C03584=1030.915,110.393,-100.515,168.841,44.081,158.264
C03585=1030.909,110.144,-100.496,168.839,44.083,158.265
C03586=1030.902,109.895,-100.475,168.837,44.085,158.265
C03587=1030.896,109.646,-100.456,168.834,44.087,158.265
C03588=1030.890,109.397,-100.436,168.831,44.089,158.265
C03589=1030.884,109.148,-100.417,168.829,44.091,158.265
C03590=1030.878,108.899,-100.397,168.826,44.093,158.265
C03591=1030.870,108.613,-100.375,168.824,44.095,158.265
C03592=1030.864,108.328,-100.352,168.821,44.097,158.266
C03593=1030.857,108.042,-100.330,168.818,44.099,158.266
C03594=1030.850,107.758,-100.307,168.815,44.101,158.266
C03595=1030.844,107.508,-100.288,168.812,44.103,158.266
C03596=1030.837,107.259,-100.268,168.811,44.105,158.266
C03597=1030.831,107.010,-100.249,168.808,44.107,158.266
C03598=1030.825,106.761,-100.229,168.806,44.109,158.267
C03599=1030.819,106.511,-100.210,168.803,44.110,158.267
C03600=1030.813,106.263,-100.191,168.800,44.112,158.267
C03601=1030.807,106.013,-100.171,168.798,44.114,158.267
C03602=1030.800,105.764,-100.151,168.795,44.115,158.267
C03603=1030.795,105.515,-100.132,168.793,44.117,158.267
C03604=1030.788,105.265,-100.113,168.791,44.119,158.267
C03605=1030.782,105.017,-100.093,168.788,44.121,158.267
C03606=1030.776,104.767,-100.074,168.786,44.123,158.268
C03607=1030.770,104.518,-100.054,168.783,44.125,158.268
C03608=1030.764,104.269,-100.035,168.781,44.127,158.268
C03609=1030.758,104.020,-100.015,168.779,44.128,158.268
C03610=1030.752,103.770,-99.996,168.776,44.130,158.268
C03611=1030.745,103.521,-99.977,168.774,44.132,158.268
C03612=1030.739,103.272,-99.957,168.771,44.134,158.268
C03613=1030.734,103.023,-99.938,168.768,44.135,158.268
C03614=1030.728,102.774,-99.918,168.767,44.137,158.269
C03615=1030.721,102.525,-99.899,168.764,44.139,158.269
C03616=1030.716,102.276,-99.880,168.762,44.141,158.269
C03617=1030.710,102.027,-99.860,168.759,44.143,158.269
C03618=1030.704,101.777,-99.841,168.756,44.145,158.269
C03619=1030.697,101.528,-99.822,168.755,44.146,158.269
C03620=1030.691,101.279,-99.802,168.752,44.148,158.269
C03621=1030.686,101.030,-99.783,168.749,44.150,158.269
C03622=1030.679,100.781,-99.764,168.747,44.151,158.270
C03623=1030.673,100.531,-99.744,168.744,44.153,158.270
C03624=1030.667,100.282,-99.725,168.743,44.155,158.270
C03625=1030.661,100.032,-99.706,168.740,44.157,158.270
C03626=1030.655,99.784,-99.686,168.737,44.159,158.270
C03627=1030.649,99.534,-99.667,168.735,44.161,158.270
C03628=1030.643,99.285,-99.648,168.732,44.163,158.270
C03629=1030.637,99.036,-99.629,168.730,44.165,158.271
C03630=1030.630,98.787,-99.610,168.728,44.166,158.271
C03631=1030.625,98.537,-99.591,168.726,44.168,158.271
C03632=1030.618,98.289,-99.572,168.723,44.170,158.271
C03633=1030.612,98.040,-99.553,168.720,44.172,158.271
C03634=1030.606,97.790,-99.534,168.718,44.174,158.271
C03635=1030.599,97.541,-99.515,168.715,44.176,158.271
C03636=1030.594,97.292,-99.496,168.714,44.178,158.272
C03637=1030.587,97.043,-99.477,168.711,44.180,158.272
C03638=1030.581,96.794,-99.457,168.708,44.181,158.272
C03639=1030.575,96.545,-99.439,168.706,44.183,158.272
C03640=1030.569,96.295,-99.420,168.703,44.185,158.272
C03641=1030.563,96.046,-99.401,168.701,44.187,158.272
C03642=1030.556,95.797,-99.382,168.699,44.189,158.273
C03643=1030.551,95.548,-99.363,168.696,44.191,158.273
C03644=1030.544,95.298,-99.344,168.694,44.193,158.273
C03645=1030.539,95.049,-99.325,168.691,44.195,158.273
C03646=1030.532,94.800,-99.306,168.689,44.197,158.273
C03647=1030.526,94.550,-99.287,168.687,44.198,158.273
C03648=1030.520,94.301,-99.269,168.684,44.200,158.273
C03649=1030.514,94.053,-99.249,168.682,44.202,158.274
C03650=1030.508,93.803,-99.230,168.679,44.204,158.274
C03651=1030.501,93.554,-99.211,168.677,44.206,158.274
C03652=1030.496,93.305,-99.192,168.675,44.208,158.274
C03653=1030.489,93.056,-99.173,168.673,44.210,158.274
C03654=1030.483,92.806,-99.154,168.670,44.211,158.274
C03655=1030.476,92.521,-99.134,168.667,44.213,158.274
C03656=1030.469,92.236,-99.112,168.665,44.215,158.275
C03657=1030.462,91.950,-99.089,168.661,44.217,158.275
C03658=1030.455,91.665,-99.068,168.659,44.219,158.275
C03659=1030.449,91.416,-99.049,168.656,44.221,158.275
C03660=1030.443,91.166,-99.030,168.654,44.223,158.275
C03661=1030.437,90.918,-99.012,168.652,44.225,158.275
C03662=1030.431,90.669,-98.993,168.649,44.227,158.275
C03663=1030.425,90.419,-98.974,168.647,44.229,158.275
C03664=1030.419,90.170,-98.955,168.644,44.231,158.276
C03665=1030.413,89.921,-98.936,168.642,44.232,158.276
C03666=1030.407,89.672,-98.917,168.640,44.234,158.276
C03667=1030.400,89.422,-98.899,168.637,44.236,158.276
C03668=1030.394,89.173,-98.881,168.635,44.238,158.276
C03669=1030.388,88.923,-98.862,168.632,44.240,158.276
C03670=1030.382,88.674,-98.843,168.631,44.242,158.277
C03671=1030.376,88.425,-98.824,168.628,44.244,158.277
C03672=1030.369,88.176,-98.806,168.625,44.245,158.277
C03673=1030.363,87.926,-98.788,168.623,44.247,158.277
C03674=1030.357,87.677,-98.769,168.620,44.249,158.277
C03675=1030.351,87.429,-98.751,168.618,44.252,158.277
C03676=1030.345,87.179,-98.731,168.616,44.254,158.278
C03677=1030.339,86.929,-98.714,168.614,44.256,158.278
C03678=1030.333,86.680,-98.695,168.611,44.257,158.278
C03679=1030.326,86.431,-98.676,168.608,44.259,158.278
C03680=1030.320,86.182,-98.658,168.606,44.261,158.278
C03681=1030.314,85.932,-98.640,168.604,44.263,158.278
C03682=1030.307,85.683,-98.621,168.602,44.265,158.278
C03683=1030.301,85.434,-98.602,168.599,44.267,158.279
C03684=1030.296,85.185,-98.583,168.597,44.269,158.279
C03685=1030.290,84.936,-98.566,168.594,44.271,158.279
C03686=1030.283,84.686,-98.547,168.591,44.273,158.279
C03687=1030.277,84.437,-98.528,168.590,44.274,158.279
C03688=1030.271,84.188,-98.510,168.587,44.276,158.279
C03689=1030.264,83.938,-98.492,168.585,44.278,158.279
C03690=1030.258,83.689,-98.473,168.582,44.280,158.280
C03691=1030.252,83.441,-98.455,168.579,44.282,158.280
C03692=1030.246,83.191,-98.437,168.578,44.284,158.280
C03693=1030.240,82.942,-98.418,168.575,44.286,158.280
C03694=1030.234,82.693,-98.399,168.573,44.288,158.280
C03695=1030.228,82.443,-98.381,168.570,44.290,158.280
C03696=1030.222,82.194,-98.363,168.567,44.291,158.280
C03697=1030.216,81.945,-98.345,168.566,44.293,158.281
C03698=1030.209,81.696,-98.326,168.563,44.295,158.281
C03699=1030.203,81.446,-98.307,168.561,44.297,158.281
C03700=1030.197,81.197,-98.290,168.558,44.299,158.281
C03701=1030.191,80.948,-98.271,168.557,44.301,158.281
C03702=1030.185,80.698,-98.253,168.554,44.303,158.281
C03703=1030.179,80.449,-98.234,168.551,44.304,158.281
C03704=1030.173,80.200,-98.215,168.549,44.306,158.282
C03705=1030.166,79.950,-98.197,168.546,44.308,158.282
C03706=1030.161,79.702,-98.179,168.545,44.310,158.282
C03707=1030.155,79.452,-98.161,168.542,44.312,158.282
C03708=1030.148,79.203,-98.143,168.539,44.314,158.282
C03709=1030.142,78.953,-98.125,168.537,44.316,158.282
C03710=1030.136,78.705,-98.106,168.535,44.318,158.282
C03711=1030.130,78.456,-98.088,168.533,44.319,158.283
C03712=1030.124,78.206,-98.070,168.530,44.321,158.283
C03713=1030.118,77.957,-98.051,168.528,44.323,158.283
C03714=1030.112,77.708,-98.033,168.525,44.325,158.283
C03715=1030.106,77.458,-98.016,168.523,44.327,158.283
C03716=1030.099,77.209,-97.997,168.521,44.329,158.283
C03717=1030.093,76.959,-97.979,168.518,44.331,158.283
C03718=1030.087,76.711,-97.961,168.516,44.333,158.284
C03719=1030.080,76.425,-97.940,168.513,44.335,158.284
C03720=1030.073,76.140,-97.919,168.511,44.337,158.284
C03721=1030.066,75.855,-97.898,168.508,44.339,158.284
C03722=1030.059,75.569,-97.878,168.505,44.342,158.284
C03723=1030.053,75.320,-97.860,168.503,44.344,158.284
C03724=1030.046,75.070,-97.842,168.501,44.346,158.285
C03725=1030.040,74.821,-97.825,168.498,44.348,158.285
C03726=1030.034,74.572,-97.806,168.495,44.349,158.285
C03727=1030.028,74.322,-97.788,168.493,44.351,158.285
C03728=1030.022,74.073,-97.771,168.490,44.353,158.285
C03729=1030.016,73.824,-97.752,168.489,44.355,158.285
C03730=1030.009,73.575,-97.735,168.486,44.357,158.285
C03731=1030.003,73.325,-97.717,168.483,44.359,158.286
C03732=1029.997,73.076,-97.698,168.481,44.361,158.286
C03733=1029.991,72.827,-97.680,168.478,44.363,158.286
C03734=1029.985,72.577,-97.662,168.477,44.365,158.286
C03735=1029.978,72.329,-97.645,168.474,44.366,158.286
C03736=1029.972,72.079,-97.627,168.471,44.368,158.286
C03737=1029.966,71.829,-97.609,168.469,44.370,158.286
C03738=1029.960,71.580,-97.591,168.466,44.372,158.287
C03739=1029.954,71.331,-97.573,168.465,44.374,158.287
C03740=1029.947,71.082,-97.555,168.462,44.376,158.287
C03741=1029.942,70.833,-97.538,168.460,44.378,158.287
C03742=1029.936,70.583,-97.520,168.457,44.380,158.287
C03743=1029.929,70.334,-97.501,168.456,44.382,158.287
C03744=1029.924,70.085,-97.484,168.453,44.384,158.288
C03745=1029.917,69.835,-97.466,168.450,44.386,158.288
C03746=1029.911,69.586,-97.448,168.448,44.388,158.288
C03747=1029.905,69.337,-97.431,168.445,44.390,158.288
C03748=1029.899,69.087,-97.412,168.444,44.392,158.288
C03749=1029.892,68.838,-97.395,168.441,44.394,158.288
C03750=1029.886,68.589,-97.377,168.439,44.395,158.288
C03751=1029.880,68.339,-97.359,168.436,44.397,158.289
C03752=1029.874,68.091,-97.342,168.433,44.399,158.289
C03753=1029.868,67.841,-97.324,168.432,44.401,158.289
C03754=1029.862,67.591,-97.306,168.429,44.403,158.289
C03755=1029.855,67.343,-97.289,168.427,44.405,158.289
C03756=1029.849,67.093,-97.271,168.424,44.407,158.289
C03757=1029.842,66.844,-97.254,168.421,44.409,158.289
C03758=1029.837,66.595,-97.236,168.419,44.411,158.290
C03759=1029.831,66.345,-97.218,168.418,44.413,158.290
C03760=1029.824,66.096,-97.201,168.415,44.415,158.290
C03761=1029.818,65.847,-97.183,168.412,44.417,158.290
C03762=1029.811,65.597,-97.166,168.410,44.419,158.290
C03763=1029.806,65.348,-97.148,168.407,44.421,158.290
C03764=1029.800,65.098,-97.130,168.406,44.423,158.290
C03765=1029.793,64.850,-97.113,168.403,44.424,158.291
C03766=1029.787,64.600,-97.095,168.400,44.426,158.291
C03767=1029.781,64.351,-97.078,168.398,44.428,158.291
C03768=1029.775,64.101,-97.060,168.395,44.430,158.291
C03769=1029.768,63.852,-97.043,168.394,44.432,158.291
C03770=1029.763,63.603,-97.026,168.391,44.434,158.291
C03771=1029.756,63.353,-97.008,168.389,44.437,158.292
C03772=1029.750,63.104,-96.991,168.386,44.439,158.292
C03773=1029.743,62.855,-96.973,168.384,44.440,158.292
C03774=1029.736,62.606,-96.956,168.381,44.442,158.292
C03775=1029.731,62.356,-96.939,168.379,44.445,158.292
C03776=1029.724,62.106,-96.922,168.377,44.447,158.292
C03777=1029.718,61.858,-96.905,168.374,44.449,158.293
C03778=1029.712,61.608,-96.887,168.372,44.451,158.293
C03779=1029.706,61.359,-96.870,168.369,44.453,158.293
C03780=1029.699,61.110,-96.853,168.367,44.455,158.293
C03781=1029.692,60.860,-96.836,168.364,44.457,158.293
C03782=1029.687,60.611,-96.818,168.362,44.459,158.293
C03783=1029.679,60.325,-96.799,168.359,44.462,158.294
C03784=1029.672,60.040,-96.778,168.357,44.464,158.294
C03785=1029.665,59.755,-96.759,168.354,44.466,158.294
C03786=1029.658,59.469,-96.739,168.351,44.468,158.294
C03787=1029.651,59.220,-96.722,168.348,44.470,158.294
C03788=1029.645,58.970,-96.706,168.347,44.472,158.294
C03789=1029.639,58.720,-96.688,168.344,44.475,158.295
C03790=1029.633,58.472,-96.671,168.342,44.477,158.295
C03791=1029.626,58.222,-96.654,168.339,44.478,158.295
C03792=1029.620,57.973,-96.637,168.337,44.480,158.295
C03793=1029.614,57.723,-96.619,168.334,44.482,158.295
C03794=1029.607,57.475,-96.602,168.332,44.484,158.295
C03795=1029.601,57.225,-96.585,168.330,44.487,158.296
C03796=1029.595,56.975,-96.568,168.328,44.489,158.296
C03797=1029.588,56.726,-96.551,168.325,44.491,158.296
C03798=1029.582,56.477,-96.534,168.322,44.492,158.296
C03799=1029.576,56.227,-96.517,168.320,44.494,158.296
C03800=1029.570,55.978,-96.500,168.318,44.496,158.296
C03801=1029.563,55.729,-96.482,168.316,44.498,158.296
C03802=1029.557,55.479,-96.466,168.313,44.501,158.297
C03803=1029.550,55.230,-96.449,168.311,44.503,158.297
C03804=1029.545,54.981,-96.431,168.308,44.505,158.297
C03805=1029.538,54.731,-96.415,168.305,44.507,158.297
C03806=1029.532,54.482,-96.398,168.303,44.508,158.297
C03807=1029.526,54.233,-96.381,168.301,44.510,158.297
C03808=1029.520,53.983,-96.363,168.299,44.512,158.297
C03809=1029.514,53.734,-96.346,168.296,44.514,158.298
C03810=1029.507,53.485,-96.329,168.294,44.517,158.298
C03811=1029.502,53.235,-96.312,168.291,44.519,158.298
C03812=1029.495,52.986,-96.295,168.290,44.520,158.298
C03813=1029.489,52.736,-96.279,168.287,44.522,158.298
C03814=1029.483,52.488,-96.262,168.284,44.524,158.298
C03815=1029.477,52.238,-96.244,168.282,44.526,158.299
C03816=1029.471,51.989,-96.228,168.279,44.528,158.299
C03817=1029.464,51.739,-96.210,168.277,44.530,158.299
C03818=1029.458,51.490,-96.194,168.275,44.532,158.299
C03819=1029.452,51.241,-96.177,168.273,44.534,158.299
C03820=1029.446,50.991,-96.160,168.270,44.536,158.299
C03821=1029.439,50.742,-96.143,168.268,44.538,158.300
C03822=1029.433,50.493,-96.127,168.265,44.540,158.300
C03823=1029.427,50.243,-96.109,168.262,44.542,158.300
C03824=1029.421,49.994,-96.092,168.261,44.544,158.300
C03825=1029.415,49.744,-96.075,168.258,44.546,158.300
C03826=1029.408,49.495,-96.058,168.256,44.548,158.300
C03827=1029.402,49.246,-96.042,168.253,44.550,158.300
C03828=1029.396,48.996,-96.024,168.251,44.552,158.300
C03829=1029.390,48.747,-96.008,168.249,44.554,158.301
C03830=1029.384,48.498,-95.991,168.246,44.555,158.301
C03831=1029.377,48.248,-95.974,168.244,44.557,158.301
C03832=1029.372,47.999,-95.957,168.241,44.559,158.301
C03833=1029.366,47.750,-95.940,168.239,44.561,158.301
C03834=1029.360,47.500,-95.924,168.237,44.563,158.301
C03835=1029.353,47.251,-95.907,168.235,44.565,158.301
C03836=1029.347,47.002,-95.890,168.232,44.567,158.302
C03837=1029.342,46.753,-95.873,168.229,44.569,158.302
C03838=1029.335,46.503,-95.856,168.227,44.571,158.302
C03839=1029.329,46.254,-95.839,168.225,44.573,158.302
C03840=1029.323,46.005,-95.823,168.223,44.575,158.302
C03841=1029.317,45.754,-95.806,168.220,44.576,158.302
C03842=1029.311,45.505,-95.789,168.217,44.578,158.302
C03843=1029.305,45.256,-95.772,168.215,44.580,158.302
C03844=1029.299,45.007,-95.755,168.213,44.582,158.303
C03845=1029.292,44.757,-95.739,168.211,44.584,158.303
C03846=1029.287,44.508,-95.722,168.208,44.586,158.303
C03847=1029.279,44.222,-95.703,168.206,44.588,158.303
C03848=1029.273,43.936,-95.684,168.203,44.591,158.303
C03849=1029.265,43.651,-95.664,168.200,44.593,158.303
C03850=1029.259,43.365,-95.646,168.197,44.595,158.303
C03851=1029.253,43.115,-95.628,168.194,44.597,158.304
C03852=1029.247,42.866,-95.612,168.193,44.598,158.304
C03853=1029.241,42.617,-95.596,168.190,44.600,158.304
C03854=1029.235,42.367,-95.579,168.188,44.602,158.304
C03855=1029.228,42.118,-95.562,168.185,44.604,158.304
C03856=1029.222,41.868,-95.546,168.183,44.606,158.304
C03857=1029.216,41.619,-95.530,168.180,44.609,158.304
C03858=1029.210,41.370,-95.513,168.178,44.611,158.305
C03859=1029.203,41.120,-95.497,168.176,44.613,158.305
C03860=1029.197,40.871,-95.480,168.173,44.614,158.305
C03861=1029.191,40.622,-95.463,168.171,44.616,158.305
C03862=1029.185,40.372,-95.447,168.168,44.618,158.305
C03863=1029.179,40.122,-95.431,168.166,44.620,158.305
C03864=1029.172,39.873,-95.415,168.163,44.622,158.305
C03865=1029.166,39.625,-95.398,168.162,44.624,158.306
C03866=1029.160,39.375,-95.382,168.159,44.626,158.306
C03867=1029.154,39.126,-95.365,168.156,44.628,158.306
C03868=1029.147,38.876,-95.349,168.154,44.630,158.306
C03869=1029.141,38.626,-95.333,168.151,44.633,158.306
C03870=1029.135,38.377,-95.316,168.149,44.634,158.306
C03871=1029.129,38.128,-95.300,168.147,44.636,158.306
C03872=1029.124,37.878,-95.284,168.145,44.638,158.307
C03873=1029.117,37.629,-95.266,168.142,44.640,158.307
C03874=1029.111,37.380,-95.250,168.140,44.642,158.307
C03875=1029.105,37.130,-95.234,168.137,44.644,158.307
C03876=1029.098,36.881,-95.218,168.134,44.646,158.307
C03877=1029.092,36.632,-95.202,168.132,44.648,158.307
C03878=1029.086,36.382,-95.185,168.130,44.650,158.307
C03879=1029.080,36.132,-95.169,168.128,44.652,158.308
C03880=1029.073,35.883,-95.154,168.125,44.654,158.308
C03881=1029.067,35.634,-95.137,168.123,44.656,158.308
C03882=1029.061,35.385,-95.121,168.120,44.658,158.308
C03883=1029.054,35.136,-95.105,168.118,44.660,158.308
C03884=1029.048,34.886,-95.089,168.115,44.662,158.308
C03885=1029.042,34.636,-95.073,168.112,44.664,158.308
C03886=1029.036,34.386,-95.057,168.110,44.667,158.309
C03887=1029.029,34.137,-95.041,168.108,44.668,158.309
C03888=1029.024,33.888,-95.025,168.106,44.670,158.309
C03889=1029.018,33.639,-95.009,168.103,44.672,158.309
C03890=1029.010,33.389,-94.993,168.101,44.674,158.309
C03891=1029.004,33.139,-94.976,168.098,44.676,158.309
C03892=1028.998,32.890,-94.960,168.096,44.678,158.309
C03893=1028.992,32.641,-94.945,168.093,44.681,158.310
C03894=1028.986,32.392,-94.928,168.091,44.683,158.310
C03895=1028.980,32.142,-94.912,168.088,44.685,158.310
C03896=1028.973,31.893,-94.897,168.086,44.687,158.310
C03897=1028.967,31.643,-94.881,168.084,44.688,158.310
C03898=1028.962,31.394,-94.865,168.081,44.690,158.310
C03899=1028.954,31.144,-94.849,168.079,44.692,158.310
C03900=1028.948,30.895,-94.832,168.076,44.694,158.311
C03901=1028.942,30.646,-94.816,168.074,44.696,158.311
C03902=1028.936,30.397,-94.800,168.071,44.699,158.311
C03903=1028.930,30.147,-94.785,168.069,44.701,158.311
C03904=1028.924,29.897,-94.769,168.067,44.703,158.311
C03905=1028.917,29.648,-94.753,168.065,44.705,158.311
C03906=1028.911,29.399,-94.737,168.062,44.707,158.311
C03907=1028.905,29.150,-94.720,168.059,44.709,158.312
C03908=1028.899,28.900,-94.705,168.057,44.710,158.312
C03909=1028.893,28.651,-94.689,168.054,44.712,158.312
C03910=1028.887,28.401,-94.673,168.052,44.714,158.312
C03911=1028.879,28.069,-94.652,168.049,44.717,158.312
C03912=1028.870,27.738,-94.631,168.046,44.720,158.312
C03913=1028.862,27.407,-94.610,168.043,44.723,158.313
C03914=1028.854,27.075,-94.589,168.039,44.726,158.313
C03915=1028.848,26.825,-94.573,168.037,44.728,158.313
C03916=1028.841,26.576,-94.558,168.034,44.729,158.313
C03917=1028.835,26.326,-94.542,168.031,44.731,158.313
C03918=1028.829,26.077,-94.526,168.029,44.733,158.313
C03919=1028.823,25.827,-94.510,168.026,44.735,158.313
C03920=1028.816,25.578,-94.495,168.024,44.737,158.314
C03921=1028.810,25.329,-94.479,168.022,44.740,158.314
C03922=1028.804,25.079,-94.463,168.020,44.742,158.314
C03923=1028.797,24.830,-94.448,168.017,44.744,158.314
C03924=1028.792,24.580,-94.432,168.015,44.746,158.314
C03925=1028.785,24.331,-94.417,168.012,44.748,158.314
C03926=1028.779,24.082,-94.400,168.009,44.750,158.314
C03927=1028.773,23.855,-94.387,168.007,44.752,158.315
C03928=1028.767,23.628,-94.373,168.005,44.753,158.315
C03929=1028.762,23.402,-94.358,168.003,44.755,158.315
C03930=1028.756,23.175,-94.344,168.000,44.757,158.315
C03931=1028.751,22.948,-94.330,167.999,44.759,158.315
C03932=1028.745,22.723,-94.316,167.996,44.761,158.315
C03933=1028.739,22.495,-94.302,167.993,44.763,158.315
C03934=1028.734,22.269,-94.288,167.992,44.765,158.316
C03935=1028.727,22.020,-94.272,167.989,44.767,158.316
C03936=1028.721,21.770,-94.256,167.987,44.769,158.316
C03937=1028.715,21.521,-94.241,167.984,44.771,158.316
C03938=1028.709,21.271,-94.225,167.982,44.773,158.316
C03939=1028.702,21.022,-94.209,167.979,44.775,158.316
C03940=1028.696,20.772,-94.195,167.977,44.777,158.316
C03941=1028.690,20.523,-94.178,167.974,44.779,158.316
C03942=1028.684,20.273,-94.163,167.971,44.781,158.317
C03943=1028.678,20.023,-94.148,167.970,44.783,158.317
C03944=1028.672,19.775,-94.132,167.967,44.785,158.317
C03945=1028.666,19.525,-94.117,167.965,44.787,158.317
C03946=1028.660,19.276,-94.101,167.962,44.789,158.317
C03947=1028.653,19.026,-94.086,167.960,44.791,158.317
C03948=1028.646,18.777,-94.071,167.957,44.793,158.317
C03949=1028.641,18.527,-94.055,167.955,44.795,158.318
C03950=1028.634,18.277,-94.040,167.952,44.797,158.318
C03951=1028.628,18.028,-94.025,167.949,44.799,158.318
C03952=1028.621,17.779,-94.010,167.947,44.801,158.318
C03953=1028.616,17.529,-93.994,167.944,44.803,158.318
C03954=1028.609,17.280,-93.978,167.942,44.806,158.318
C03955=1028.603,17.030,-93.963,167.939,44.808,158.318
C03956=1028.598,16.781,-93.948,167.937,44.810,158.319
C03957=1028.591,16.532,-93.933,167.934,44.812,158.319
C03958=1028.585,16.282,-93.918,167.932,44.814,158.319
C03959=1028.578,16.032,-93.903,167.929,44.816,158.319
C03960=1028.572,15.783,-93.886,167.928,44.817,158.319
C03961=1028.566,15.533,-93.872,167.925,44.820,158.319
C03962=1028.559,15.284,-93.857,167.923,44.822,158.319
C03963=1028.553,15.036,-93.841,167.920,44.824,158.320
C03964=1028.548,14.786,-93.826,167.917,44.826,158.320
C03965=1028.541,14.536,-93.811,167.915,44.828,158.320
C03966=1028.535,14.286,-93.796,167.912,44.830,158.320
C03967=1028.528,14.037,-93.780,167.910,44.832,158.320
C03968=1028.523,13.787,-93.765,167.907,44.834,158.320
C03969=1028.516,13.538,-93.750,167.905,44.837,158.320
C03970=1028.510,13.289,-93.735,167.902,44.839,158.320
C03971=1028.504,13.039,-93.720,167.900,44.840,158.321
C03972=1028.498,12.789,-93.705,167.897,44.842,158.321
C03973=1028.491,12.540,-93.690,167.895,44.845,158.321
C03974=1028.485,12.291,-93.675,167.892,44.847,158.321
C03975=1028.477,12.006,-93.659,167.890,44.849,158.321
C03976=1028.470,11.721,-93.641,167.886,44.852,158.321
C03977=1028.463,11.437,-93.624,167.884,44.855,158.322
C03978=1028.456,11.153,-93.607,167.880,44.857,158.322
C03979=1028.449,10.903,-93.592,167.878,44.859,158.322
C03980=1028.443,10.653,-93.577,167.875,44.861,158.322
C03981=1028.436,10.404,-93.562,167.873,44.863,158.322
C03982=1028.430,10.154,-93.547,167.870,44.865,158.322
C03983=1028.424,9.905,-93.533,167.868,44.867,158.322
C03984=1028.418,9.655,-93.518,167.865,44.869,158.323
C03985=1028.412,9.406,-93.503,167.863,44.872,158.323
C03986=1028.405,9.156,-93.488,167.860,44.874,158.323
C03987=1028.399,8.907,-93.473,167.858,44.876,158.323
C03988=1028.393,8.657,-93.459,167.855,44.878,158.323
C03989=1028.387,8.408,-93.444,167.852,44.880,158.323
C03990=1028.380,8.158,-93.429,167.850,44.882,158.323
C03991=1028.374,7.909,-93.414,167.847,44.884,158.324
C03992=1028.368,7.659,-93.399,167.845,44.886,158.324
C03993=1028.362,7.410,-93.384,167.842,44.888,158.324
C03994=1028.355,7.160,-93.369,167.840,44.890,158.324
C03995=1028.350,6.911,-93.355,167.837,44.893,158.324
C03996=1028.343,6.662,-93.340,167.835,44.895,158.324
C03997=1028.337,6.412,-93.325,167.832,44.897,158.324
C03998=1028.330,6.162,-93.310,167.830,44.899,158.325
C03999=1028.325,5.913,-93.295,167.827,44.901,158.325
C04000=1028.318,5.664,-93.280,167.824,44.903,158.325
C04001=1028.312,5.414,-93.265,167.822,44.906,158.325
C04002=1028.306,5.165,-93.251,167.820,44.908,158.325
C04003=1028.300,4.915,-93.236,167.817,44.910,158.325
C04004=1028.293,4.666,-93.221,167.814,44.912,158.325
C04005=1028.287,4.416,-93.206,167.812,44.914,158.325
C04006=1028.281,4.166,-93.192,167.809,44.915,158.326
C04007=1028.275,3.917,-93.177,167.807,44.918,158.326
C04008=1028.269,3.667,-93.162,167.804,44.920,158.326
C04009=1028.263,3.418,-93.148,167.802,44.922,158.326
C04010=1028.256,3.169,-93.133,167.799,44.924,158.326
C04011=1028.249,2.919,-93.118,167.797,44.926,158.326
C04012=1028.244,2.670,-93.104,167.794,44.928,158.326
C04013=1028.238,2.420,-93.089,167.791,44.930,158.326
C04014=1028.232,2.171,-93.075,167.789,44.932,158.327
C04015=1028.225,1.921,-93.060,167.787,44.935,158.327
C04016=1028.219,1.672,-93.045,167.784,44.937,158.327
C04017=1028.213,1.423,-93.030,167.781,44.939,158.327
C04018=1028.207,1.172,-93.016,167.779,44.941,158.327
C04019=1028.201,0.923,-93.001,167.776,44.943,158.327
C04020=1028.195,0.674,-92.987,167.774,44.945,158.327
C04021=1028.189,0.424,-92.972,167.771,44.947,158.327
C04022=1028.183,0.175,-92.957,167.768,44.949,158.328
C04023=1028.177,-0.075,-92.943,167.766,44.951,158.328
C04024=1028.170,-0.325,-92.928,167.763,44.952,158.328
C04025=1028.165,-0.574,-92.913,167.761,44.954,158.328
C04026=1028.157,-0.823,-92.899,167.758,44.957,158.328
C04027=1028.152,-1.073,-92.885,167.756,44.959,158.328
C04028=1028.146,-1.322,-92.870,167.753,44.961,158.328
C04029=1028.140,-1.571,-92.856,167.751,44.963,158.328
C04030=1028.134,-1.821,-92.841,167.748,44.965,158.329
C04031=1028.127,-2.071,-92.826,167.746,44.967,158.329
C04032=1028.122,-2.320,-92.812,167.743,44.969,158.329
C04033=1028.115,-2.570,-92.797,167.740,44.971,158.329
C04034=1028.110,-2.819,-92.783,167.738,44.973,158.329
C04035=1028.103,-3.069,-92.768,167.735,44.975,158.329
C04036=1028.098,-3.318,-92.754,167.733,44.977,158.329
C04037=1028.091,-3.568,-92.739,167.730,44.979,158.329
C04038=1028.086,-3.817,-92.725,167.727,44.981,158.329
C04039=1028.078,-4.100,-92.709,167.725,44.984,158.330
C04040=1028.071,-4.382,-92.692,167.722,44.986,158.330
C04041=1028.064,-4.665,-92.677,167.719,44.988,158.330
C04042=1028.057,-4.948,-92.661,167.716,44.991,158.330
C04043=1028.050,-5.197,-92.647,167.713,44.993,158.330
C04044=1028.044,-5.447,-92.632,167.711,44.995,158.330
C04045=1028.038,-5.696,-92.618,167.708,44.997,158.331
C04046=1028.032,-5.946,-92.604,167.706,44.999,158.331
C04047=1028.026,-6.195,-92.590,167.703,45.002,158.331
C04048=1028.019,-6.445,-92.576,167.701,45.004,158.331
C04049=1028.013,-6.694,-92.561,167.698,45.006,158.331
C04050=1028.006,-6.944,-92.548,167.696,45.008,158.331
C04051=1028.001,-7.194,-92.534,167.693,45.010,158.331
C04052=1027.995,-7.443,-92.519,167.691,45.013,158.332
C04053=1027.988,-7.693,-92.506,167.688,45.015,158.332
C04054=1027.982,-7.942,-92.491,167.684,45.017,158.332
C04055=1027.976,-8.191,-92.477,167.682,45.019,158.332
C04056=1027.969,-8.441,-92.462,167.680,45.021,158.332
C04057=1027.963,-8.690,-92.449,167.677,45.023,158.332
C04058=1027.957,-8.941,-92.435,167.674,45.025,158.332
C04059=1027.951,-9.190,-92.420,167.672,45.027,158.332
C04060=1027.944,-9.440,-92.407,167.669,45.029,158.332
C04061=1027.939,-9.689,-92.393,167.667,45.032,158.333
C04062=1027.932,-9.938,-92.378,167.664,45.034,158.333
C04063=1027.926,-10.188,-92.365,167.662,45.036,158.333
C04064=1027.920,-10.437,-92.351,167.659,45.038,158.333
C04065=1027.914,-10.687,-92.336,167.657,45.040,158.333
C04066=1027.908,-10.936,-92.323,167.653,45.042,158.333
C04067=1027.901,-11.186,-92.308,167.651,45.045,158.333
C04068=1027.896,-11.435,-92.294,167.648,45.047,158.334
C04069=1027.889,-11.685,-92.281,167.645,45.049,158.334
C04070=1027.883,-11.935,-92.267,167.643,45.051,158.334
C04071=1027.877,-12.184,-92.253,167.640,45.053,158.334
C04072=1027.871,-12.434,-92.239,167.638,45.055,158.334
C04073=1027.865,-12.683,-92.225,167.635,45.057,158.334
C04074=1027.858,-12.933,-92.210,167.633,45.059,158.334
C04075=1027.852,-13.182,-92.197,167.630,45.061,158.334
C04076=1027.846,-13.432,-92.183,167.628,45.063,158.335
C04077=1027.840,-13.682,-92.170,167.625,45.065,158.335
C04078=1027.834,-13.931,-92.155,167.622,45.068,158.335
C04079=1027.828,-14.180,-92.141,167.619,45.070,158.335
C04080=1027.822,-14.430,-92.128,167.617,45.072,158.335
C04081=1027.816,-14.680,-92.114,167.614,45.074,158.335
C04082=1027.809,-14.930,-92.100,167.611,45.076,158.335
C04083=1027.804,-15.179,-92.085,167.609,45.078,158.335
C04084=1027.797,-15.428,-92.072,167.606,45.080,158.335
C04085=1027.791,-15.678,-92.058,167.604,45.082,158.336
C04086=1027.785,-15.927,-92.045,167.601,45.085,158.336
C04087=1027.779,-16.177,-92.031,167.599,45.087,158.336
C04088=1027.773,-16.427,-92.017,167.595,45.089,158.336
C04089=1027.767,-16.676,-92.004,167.593,45.091,158.336
C04090=1027.760,-16.926,-91.991,167.590,45.094,158.336
C04091=1027.753,-17.176,-91.977,167.588,45.096,158.336
C04092=1027.748,-17.425,-91.963,167.585,45.098,158.337
C04093=1027.742,-17.674,-91.950,167.583,45.100,158.337
C04094=1027.735,-17.924,-91.936,167.579,45.103,158.337
C04095=1027.729,-18.173,-91.922,167.577,45.105,158.337
C04096=1027.723,-18.423,-91.908,167.574,45.107,158.337
C04097=1027.716,-18.672,-91.895,167.572,45.109,158.337
C04098=1027.710,-18.922,-91.882,167.569,45.111,158.337
C04099=1027.704,-19.171,-91.868,167.567,45.113,158.337
C04100=1027.698,-19.421,-91.854,167.564,45.115,158.338
C04101=1027.691,-19.671,-91.841,167.560,45.118,158.338
C04102=1027.685,-19.920,-91.827,167.558,45.120,158.338
C04103=1027.679,-20.202,-91.812,167.556,45.122,158.338
C04104=1027.672,-20.483,-91.797,167.552,45.125,158.338
C04105=1027.665,-20.763,-91.782,167.550,45.127,158.338
C04106=1027.658,-21.044,-91.767,167.546,45.130,158.338
C04107=1027.652,-21.294,-91.754,167.544,45.132,158.339
C04108=1027.645,-21.544,-91.740,167.541,45.134,158.339
C04109=1027.640,-21.793,-91.726,167.539,45.136,158.339
C04110=1027.633,-22.043,-91.713,167.535,45.139,158.339
C04111=1027.627,-22.292,-91.700,167.533,45.141,158.339
C04112=1027.620,-22.542,-91.686,167.530,45.143,158.339
C04113=1027.615,-22.791,-91.672,167.527,45.145,158.339
C04114=1027.609,-23.041,-91.660,167.525,45.147,158.339
C04115=1027.603,-23.290,-91.646,167.523,45.150,158.340
C04116=1027.596,-23.540,-91.633,167.519,45.152,158.340
C04117=1027.590,-23.790,-91.619,167.516,45.154,158.340
C04118=1027.584,-24.039,-91.606,167.514,45.156,158.340
C04119=1027.578,-24.289,-91.592,167.511,45.158,158.340
C04120=1027.572,-24.538,-91.579,167.509,45.161,158.340
C04121=1027.567,-24.788,-91.566,167.506,45.163,158.340
C04122=1027.560,-25.038,-91.552,167.504,45.165,158.340
C04123=1027.554,-25.287,-91.539,167.500,45.167,158.340
C04124=1027.547,-25.537,-91.526,167.498,45.169,158.340
C04125=1027.542,-25.786,-91.512,167.495,45.171,158.341
C04126=1027.536,-26.036,-91.499,167.493,45.173,158.341
C04127=1027.530,-26.285,-91.486,167.490,45.175,158.341
C04128=1027.524,-26.534,-91.473,167.488,45.177,158.341
C04129=1027.517,-26.785,-91.458,167.484,45.180,158.341
C04130=1027.511,-27.034,-91.445,167.481,45.182,158.341
C04131=1027.505,-27.284,-91.433,167.479,45.184,158.341
C04132=1027.499,-27.533,-91.419,167.476,45.186,158.342
C04133=1027.493,-27.782,-91.406,167.474,45.188,158.342
C04134=1027.487,-28.032,-91.394,167.470,45.191,158.342
C04135=1027.481,-28.282,-91.380,167.468,45.193,158.342
C04136=1027.474,-28.532,-91.367,167.465,45.195,158.342
C04137=1027.468,-28.781,-91.354,167.463,45.197,158.342
C04138=1027.462,-29.031,-91.341,167.461,45.200,158.342
C04139=1027.456,-29.281,-91.328,167.457,45.202,158.342
C04140=1027.450,-29.530,-91.315,167.454,45.204,158.342
C04141=1027.444,-29.780,-91.302,167.452,45.207,158.343
C04142=1027.438,-30.029,-91.289,167.449,45.209,158.343
C04143=1027.431,-30.278,-91.276,167.446,45.211,158.343
C04144=1027.425,-30.529,-91.263,167.443,45.213,158.343
C04145=1027.419,-30.778,-91.250,167.441,45.216,158.343
C04146=1027.413,-31.028,-91.237,167.438,45.218,158.343
C04147=1027.406,-31.277,-91.224,167.436,45.220,158.343
C04148=1027.400,-31.527,-91.212,167.432,45.223,158.344
C04149=1027.394,-31.776,-91.199,167.430,45.225,158.344
C04150=1027.388,-32.026,-91.186,167.427,45.227,158.344
C04151=1027.382,-32.275,-91.173,167.425,45.229,158.344
C04152=1027.376,-32.525,-91.160,167.421,45.232,158.344
C04153=1027.369,-32.774,-91.147,167.419,45.234,158.344
C04154=1027.363,-33.024,-91.134,167.416,45.236,158.344
C04155=1027.357,-33.274,-91.121,167.414,45.238,158.344
C04156=1027.351,-33.523,-91.109,167.411,45.240,158.345
C04157=1027.345,-33.773,-91.095,167.408,45.243,158.345
C04158=1027.339,-34.023,-91.083,167.405,45.245,158.345
C04159=1027.333,-34.272,-91.070,167.403,45.247,158.345
C04160=1027.327,-34.522,-91.057,167.400,45.249,158.345
C04161=1027.321,-34.771,-91.044,167.397,45.251,158.345
C04162=1027.315,-35.021,-91.031,167.394,45.254,158.345
C04163=1027.309,-35.271,-91.019,167.392,45.256,158.345
C04164=1027.303,-35.520,-91.005,167.389,45.258,158.346
C04165=1027.296,-35.770,-90.993,167.386,45.260,158.346
C04166=1027.290,-36.019,-90.980,167.383,45.262,158.346
C04167=1027.283,-36.300,-90.966,167.381,45.265,158.346
C04168=1027.276,-36.580,-90.951,167.377,45.267,158.346
C04169=1027.270,-36.860,-90.938,167.374,45.270,158.346
C04170=1027.263,-37.140,-90.923,167.371,45.272,158.346
C04171=1027.257,-37.390,-90.910,167.368,45.275,158.346
C04172=1027.251,-37.639,-90.897,167.365,45.277,158.346
C04173=1027.245,-37.889,-90.884,167.363,45.279,158.347
C04174=1027.239,-38.139,-90.872,167.360,45.281,158.347
C04175=1027.233,-38.388,-90.859,167.358,45.283,158.347
C04176=1027.227,-38.638,-90.846,167.354,45.285,158.347
C04177=1027.221,-38.888,-90.833,167.352,45.288,158.347
C04178=1027.214,-39.137,-90.822,167.349,45.290,158.347
C04179=1027.208,-39.386,-90.808,167.346,45.292,158.347
C04180=1027.202,-39.636,-90.796,167.343,45.295,158.347
C04181=1027.197,-39.886,-90.784,167.341,45.297,158.347
C04182=1027.190,-40.135,-90.772,167.338,45.299,158.348
C04183=1027.184,-40.385,-90.759,167.335,45.302,158.348
C04184=1027.178,-40.635,-90.746,167.332,45.304,158.348
C04185=1027.172,-40.884,-90.734,167.330,45.307,158.348
C04186=1027.166,-41.134,-90.721,167.326,45.309,158.348
C04187=1027.160,-41.384,-90.709,167.324,45.311,158.348
C04188=1027.153,-41.633,-90.697,167.321,45.314,158.348
C04189=1027.147,-41.883,-90.684,167.319,45.316,158.349
C04190=1027.140,-42.133,-90.672,167.315,45.318,158.349
C04191=1027.135,-42.382,-90.660,167.313,45.321,158.349
C04192=1027.129,-42.631,-90.647,167.310,45.323,158.349
C04193=1027.122,-42.881,-90.635,167.307,45.325,158.349
C04194=1027.116,-43.131,-90.622,167.304,45.328,158.349
C04195=1027.111,-43.380,-90.610,167.302,45.330,158.349
C04196=1027.104,-43.630,-90.598,167.298,45.332,158.349
C04197=1027.098,-43.880,-90.585,167.296,45.335,158.350
C04198=1027.093,-44.129,-90.573,167.293,45.337,158.350
C04199=1027.086,-44.379,-90.561,167.291,45.339,158.350
C04200=1027.080,-44.629,-90.548,167.287,45.342,158.350
C04201=1027.074,-44.878,-90.536,167.285,45.344,158.350
C04202=1027.068,-45.128,-90.524,167.282,45.346,158.350
C04203=1027.062,-45.377,-90.512,167.279,45.348,158.350
C04204=1027.056,-45.627,-90.499,167.276,45.350,158.350
C04205=1027.050,-45.877,-90.487,167.274,45.353,158.350
C04206=1027.044,-46.127,-90.475,167.270,45.355,158.351
C04207=1027.037,-46.376,-90.463,167.268,45.357,158.351
C04208=1027.032,-46.625,-90.451,167.265,45.359,158.351
C04209=1027.026,-46.875,-90.438,167.263,45.361,158.351
C04210=1027.019,-47.125,-90.426,167.259,45.364,158.351
C04211=1027.013,-47.375,-90.413,167.257,45.366,158.351
C04212=1027.008,-47.624,-90.401,167.254,45.368,158.351
C04213=1027.001,-47.873,-90.389,167.251,45.371,158.351
C04214=1026.995,-48.123,-90.377,167.248,45.373,158.352
C04215=1026.989,-48.373,-90.365,167.246,45.375,158.352
C04216=1026.984,-48.622,-90.353,167.242,45.378,158.352
C04217=1026.978,-48.872,-90.340,167.240,45.380,158.352
C04218=1026.971,-49.122,-90.329,167.237,45.382,158.352
C04219=1026.965,-49.372,-90.316,167.234,45.385,158.352
C04220=1026.960,-49.621,-90.304,167.231,45.387,158.352
C04221=1026.953,-49.871,-90.292,167.229,45.389,158.352
C04222=1026.948,-50.121,-90.280,167.226,45.391,158.352
C04223=1026.941,-50.369,-90.268,167.223,45.394,158.352
C04224=1026.936,-50.619,-90.255,167.220,45.396,158.353
C04225=1026.929,-50.870,-90.244,167.218,45.398,158.353
C04226=1026.923,-51.119,-90.232,167.214,45.401,158.353
C04227=1026.917,-51.368,-90.220,167.212,45.403,158.353
C04228=1026.911,-51.618,-90.209,167.208,45.406,158.353
C04229=1026.904,-51.868,-90.197,167.206,45.408,158.353
C04230=1026.898,-52.118,-90.184,167.203,45.411,158.354
C04231=1026.892,-52.398,-90.172,167.200,45.413,158.354
C04232=1026.884,-52.679,-90.158,167.197,45.416,158.354
C04233=1026.878,-52.960,-90.145,167.193,45.419,158.354
C04234=1026.871,-53.240,-90.132,167.190,45.422,158.354
C04235=1026.864,-53.489,-90.120,167.187,45.424,158.354
C04236=1026.858,-53.739,-90.109,167.184,45.427,158.354
C04237=1026.853,-53.989,-90.097,167.181,45.429,158.354
C04238=1026.846,-54.239,-90.085,167.179,45.432,158.355
C04239=1026.840,-54.488,-90.073,167.175,45.434,158.355
C04240=1026.834,-54.737,-90.062,167.173,45.437,158.355
C04241=1026.828,-54.988,-90.050,167.170,45.439,158.355
C04242=1026.821,-55.237,-90.038,167.167,45.442,158.355
C04243=1026.816,-55.487,-90.027,167.165,45.444,158.355
C04244=1026.809,-55.736,-90.015,167.161,45.447,158.355
C04245=1026.803,-55.986,-90.004,167.159,45.449,158.356
C04246=1026.797,-56.236,-89.992,167.155,45.452,158.356
C04247=1026.791,-56.485,-89.980,167.153,45.454,158.356
C04248=1026.785,-56.735,-89.969,167.150,45.456,158.356
C04249=1026.778,-56.984,-89.957,167.147,45.458,158.356
C04250=1026.773,-57.234,-89.946,167.145,45.461,158.356
C04251=1026.767,-57.484,-89.933,167.141,45.463,158.356
C04252=1026.760,-57.734,-89.922,167.139,45.466,158.357
C04253=1026.754,-57.983,-89.911,167.135,45.468,158.357
C04254=1026.748,-58.233,-89.899,167.133,45.471,158.357
C04255=1026.743,-58.482,-89.887,167.130,45.473,158.357
C04256=1026.736,-58.732,-89.876,167.127,45.476,158.357
C04257=1026.731,-58.982,-89.865,167.124,45.478,158.357
C04258=1026.724,-59.231,-89.853,167.121,45.480,158.357
C04259=1026.718,-59.482,-89.842,167.118,45.483,158.357
C04260=1026.712,-59.731,-89.830,167.116,45.485,158.357
C04261=1026.706,-59.981,-89.818,167.112,45.488,158.358
C04262=1026.700,-60.230,-89.807,167.110,45.490,158.358
C04263=1026.694,-60.480,-89.796,167.107,45.493,158.358
C04264=1026.688,-60.730,-89.785,167.104,45.495,158.358
C04265=1026.682,-60.979,-89.772,167.101,45.498,158.358
C04266=1026.676,-61.229,-89.761,167.098,45.500,158.358
C04267=1026.669,-61.478,-89.749,167.096,45.503,158.358
C04268=1026.664,-61.728,-89.738,167.092,45.505,158.358
C04269=1026.657,-61.978,-89.727,167.090,45.507,158.359
C04270=1026.651,-62.227,-89.716,167.086,45.510,158.359
C04271=1026.646,-62.478,-89.704,167.084,45.512,158.359
C04272=1026.640,-62.727,-89.693,167.081,45.515,158.359
C04273=1026.633,-62.977,-89.681,167.078,45.517,158.359
C04274=1026.628,-63.226,-89.670,167.075,45.520,158.359
C04275=1026.622,-63.476,-89.659,167.072,45.522,158.359
C04276=1026.615,-63.725,-89.647,167.069,45.524,158.359
C04277=1026.610,-63.975,-89.636,167.067,45.527,158.360
C04278=1026.604,-64.225,-89.625,167.063,45.529,158.360
C04279=1026.598,-64.475,-89.614,167.061,45.532,158.360
C04280=1026.592,-64.724,-89.602,167.058,45.534,158.360
C04281=1026.586,-64.974,-89.591,167.055,45.536,158.360
C04282=1026.580,-65.223,-89.580,167.052,45.539,158.360
C04283=1026.574,-65.474,-89.568,167.049,45.541,158.360
C04284=1026.568,-65.723,-89.557,167.047,45.544,158.360
C04285=1026.562,-65.973,-89.545,167.043,45.546,158.360
C04286=1026.556,-66.222,-89.534,167.041,45.548,158.361
C04287=1026.551,-66.472,-89.524,167.037,45.551,158.361
C04288=1026.544,-66.721,-89.512,167.035,45.553,158.361
C04289=1026.539,-66.971,-89.500,167.032,45.556,158.361
C04290=1026.533,-67.221,-89.489,167.029,45.558,158.361
///RCONF 1,0,0,1,0,0,0,0,0,0,0,0,0,0,0,0,0,0,0,0,0,0,0,0
C04291=1026.527,-67.471,-89.478,167.026,45.560,158.361
C04292=1026.521,-67.720,-89.467,167.023,45.563,158.361
C04293=1026.515,-67.970,-89.456,167.020,45.565,158.361
C04294=1026.509,-68.219,-89.444,167.017,45.568,158.362
C04295=1026.503,-68.501,-89.432,167.014,45.570,158.362
C04296=1026.496,-68.783,-89.420,167.011,45.573,158.362
C04297=1026.490,-69.065,-89.407,167.008,45.576,158.362
C04298=1026.483,-69.346,-89.394,167.004,45.578,158.362
C04299=1026.477,-69.596,-89.382,167.002,45.581,158.362
C04300=1026.471,-69.846,-89.371,166.998,45.583,158.362
C04301=1026.465,-70.095,-89.361,166.996,45.585,158.362
C04302=1026.460,-70.345,-89.350,166.992,45.588,158.362
C04303=1026.453,-70.595,-89.339,166.990,45.590,158.363
C04304=1026.447,-70.845,-89.328,166.987,45.592,158.363
C04305=1026.442,-71.094,-89.316,166.984,45.595,158.363
C04306=1026.436,-71.345,-89.305,166.981,45.597,158.363
C04307=1026.430,-71.594,-89.294,166.978,45.599,158.363
C04308=1026.425,-71.844,-89.283,166.975,45.602,158.363
C04309=1026.419,-72.093,-89.272,166.973,45.604,158.363
C04310=1026.413,-72.343,-89.261,166.969,45.607,158.363
C04311=1026.407,-72.593,-89.250,166.967,45.609,158.363
C04312=1026.401,-72.842,-89.239,166.963,45.611,158.363
C04313=1026.395,-73.092,-89.228,166.961,45.614,158.364
C04314=1026.390,-73.342,-89.217,166.957,45.616,158.364
C04315=1026.384,-73.592,-89.206,166.955,45.618,158.364
C04316=1026.378,-73.841,-89.195,166.952,45.621,158.364
C04317=1026.373,-74.091,-89.184,166.949,45.623,158.364
C04318=1026.367,-74.340,-89.173,166.946,45.626,158.364
C04319=1026.360,-74.590,-89.162,166.943,45.628,158.364
C04320=1026.355,-74.840,-89.151,166.940,45.631,158.364
C04321=1026.349,-75.089,-89.140,166.937,45.633,158.365
C04322=1026.343,-75.339,-89.130,166.935,45.636,158.365
C04323=1026.336,-75.589,-89.119,166.931,45.638,158.365
C04324=1026.331,-75.839,-89.108,166.929,45.641,158.365
C04325=1026.325,-76.088,-89.097,166.925,45.643,158.365
C04326=1026.319,-76.338,-89.087,166.923,45.646,158.365
C04327=1026.314,-76.588,-89.076,166.919,45.648,158.365
C04328=1026.307,-76.837,-89.066,166.917,45.651,158.365
C04329=1026.301,-77.087,-89.055,166.913,45.653,158.365
C04330=1026.295,-77.337,-89.044,166.911,45.656,158.366
C04331=1026.290,-77.586,-89.033,166.908,45.658,158.366
C04332=1026.284,-77.836,-89.023,166.905,45.661,158.366
C04333=1026.278,-78.086,-89.013,166.902,45.663,158.366
C04334=1026.272,-78.335,-89.002,166.899,45.666,158.366
C04335=1026.266,-78.586,-88.991,166.896,45.668,158.366
C04336=1026.260,-78.835,-88.980,166.893,45.671,158.366
C04337=1026.254,-79.085,-88.970,166.890,45.673,158.366
C04338=1026.249,-79.334,-88.959,166.888,45.676,158.367
C04339=1026.242,-79.584,-88.949,166.884,45.678,158.367
C04340=1026.237,-79.834,-88.938,166.882,45.681,158.367
C04341=1026.231,-80.084,-88.928,166.879,45.683,158.367
C04342=1026.226,-80.333,-88.917,166.876,45.686,158.367
C04343=1026.218,-80.583,-88.907,166.872,45.689,158.367
C04344=1026.213,-80.833,-88.896,166.870,45.691,158.367
C04345=1026.207,-81.082,-88.886,166.867,45.694,158.368
C04346=1026.201,-81.333,-88.876,166.864,45.697,158.368
C04347=1026.195,-81.582,-88.866,166.861,45.699,158.368
C04348=1026.189,-81.832,-88.856,166.858,45.702,158.368
C04349=1026.183,-82.081,-88.845,166.855,45.705,158.368
C04350=1026.177,-82.331,-88.835,166.851,45.707,158.368
C04351=1026.172,-82.581,-88.824,166.849,45.710,158.368
C04352=1026.165,-82.830,-88.815,166.846,45.713,158.369
C04353=1026.160,-83.080,-88.804,166.843,45.715,158.369
C04354=1026.153,-83.330,-88.794,166.840,45.718,158.369
C04355=1026.147,-83.580,-88.783,166.838,45.721,158.369
C04356=1026.141,-83.830,-88.773,166.834,45.723,158.369
C04357=1026.135,-84.079,-88.762,166.832,45.726,158.369
C04358=1026.129,-84.329,-88.753,166.828,45.729,158.369
C04359=1026.123,-84.613,-88.741,166.825,45.732,158.370
C04360=1026.116,-84.896,-88.730,166.822,45.735,158.370
C04361=1026.109,-85.180,-88.718,166.818,45.738,158.370
C04362=1026.103,-85.464,-88.706,166.815,45.741,158.370
C04363=1026.097,-85.714,-88.697,166.811,45.743,158.370
C04364=1026.091,-85.964,-88.686,166.809,45.746,158.370
C04365=1026.085,-86.214,-88.676,166.806,45.749,158.370
C04366=1026.079,-86.463,-88.665,166.803,45.751,158.370
C04367=1026.073,-86.713,-88.656,166.800,45.754,158.371
C04368=1026.067,-86.963,-88.646,166.796,45.757,158.371
C04369=1026.061,-87.212,-88.635,166.794,45.759,158.371
C04370=1026.056,-87.462,-88.625,166.791,45.762,158.371
C04371=1026.049,-87.712,-88.616,166.788,45.764,158.371
C04372=1026.044,-87.961,-88.605,166.785,45.767,158.371
C04373=1026.037,-88.211,-88.595,166.782,45.769,158.371
C04374=1026.032,-88.461,-88.585,166.779,45.772,158.372
C04375=1026.026,-88.711,-88.575,166.776,45.774,158.372
C04376=1026.020,-88.961,-88.564,166.773,45.777,158.372
C04377=1026.014,-89.210,-88.555,166.770,45.780,158.372
C04378=1026.009,-89.460,-88.545,166.767,45.782,158.372
C04379=1026.003,-89.709,-88.535,166.764,45.785,158.372
C04380=1025.997,-89.959,-88.525,166.761,45.787,158.372
C04381=1025.991,-90.209,-88.515,166.758,45.790,158.372
C04382=1025.986,-90.459,-88.505,166.756,45.793,158.373
C04383=1025.979,-90.708,-88.495,166.752,45.795,158.373
C04384=1025.974,-90.958,-88.485,166.750,45.798,158.373
C04385=1025.968,-91.208,-88.475,166.746,45.800,158.373
C04386=1025.962,-91.458,-88.465,166.743,45.803,158.373
C04387=1025.957,-91.707,-88.456,166.741,45.806,158.373
C04388=1025.951,-91.957,-88.445,166.737,45.808,158.373
C04389=1025.945,-92.207,-88.435,166.735,45.811,158.373
C04390=1025.939,-92.457,-88.425,166.731,45.813,158.373
C04391=1025.933,-92.707,-88.415,166.729,45.816,158.374
C04392=1025.928,-92.957,-88.405,166.725,45.819,158.374
C04393=1025.922,-93.206,-88.396,166.723,45.821,158.374
C04394=1025.916,-93.455,-88.385,166.720,45.824,158.374
C04395=1025.910,-93.705,-88.376,166.716,45.827,158.374
C04396=1025.905,-93.955,-88.365,166.714,45.829,158.374
C04397=1025.898,-94.205,-88.356,166.710,45.832,158.374
C04398=1025.894,-94.454,-88.346,166.708,45.834,158.374
C04399=1025.887,-94.704,-88.337,166.704,45.837,158.375
C04400=1025.882,-94.954,-88.326,166.702,45.840,158.375
C04401=1025.876,-95.204,-88.317,166.699,45.842,158.375
C04402=1025.870,-95.454,-88.307,166.696,45.845,158.375
C04403=1025.865,-95.703,-88.297,166.693,45.847,158.375
C04404=1025.859,-95.953,-88.287,166.690,45.850,158.375
C04405=1025.853,-96.203,-88.277,166.687,45.852,158.375
C04406=1025.847,-96.452,-88.267,166.683,45.855,158.375
C04407=1025.842,-96.702,-88.258,166.681,45.858,158.376
C04408=1025.836,-96.952,-88.248,166.678,45.860,158.376
C04409=1025.830,-97.202,-88.238,166.675,45.863,158.376
C04410=1025.825,-97.451,-88.229,166.672,45.866,158.376
C04411=1025.819,-97.701,-88.219,166.669,45.868,158.376
C04412=1025.813,-97.951,-88.209,166.666,45.871,158.376
C04413=1025.807,-98.201,-88.200,166.663,45.874,158.376
C04414=1025.802,-98.450,-88.191,166.660,45.876,158.376
C04415=1025.796,-98.700,-88.181,166.657,45.879,158.377
C04416=1025.790,-98.950,-88.171,166.654,45.882,158.377
C04417=1025.784,-99.200,-88.162,166.651,45.885,158.377
C04418=1025.778,-99.449,-88.152,166.648,45.887,158.377
C04419=1025.772,-99.699,-88.143,166.645,45.890,158.377
C04420=1025.767,-99.950,-88.133,166.642,45.893,158.377
C04421=1025.762,-100.199,-88.124,166.639,45.896,158.377
C04422=1025.755,-100.448,-88.115,166.636,45.898,158.378
C04423=1025.749,-100.735,-88.104,166.633,45.902,158.378
C04424=1025.742,-101.020,-88.093,166.630,45.905,158.378
C04425=1025.735,-101.307,-88.082,166.625,45.908,158.378
C04426=1025.729,-101.592,-88.072,166.622,45.911,158.378
C04427=1025.723,-101.843,-88.062,166.620,45.914,158.378
C04428=1025.718,-102.092,-88.052,166.616,45.917,158.379
C04429=1025.712,-102.342,-88.044,166.613,45.919,158.379
C04430=1025.706,-102.592,-88.034,166.610,45.922,158.379
C04431=1025.700,-102.841,-88.025,166.607,45.925,158.379
C04432=1025.694,-103.091,-88.015,166.605,45.928,158.379
C04433=1025.689,-103.342,-88.006,166.601,45.930,158.379
C04434=1025.683,-103.591,-87.997,166.598,45.933,158.379
C04435=1025.677,-103.840,-87.987,166.596,45.936,158.380
C04436=1025.672,-104.090,-87.979,166.592,45.939,158.380
C04437=1025.666,-104.340,-87.969,166.590,45.941,158.380
C04438=1025.659,-104.590,-87.959,166.586,45.944,158.380
C04439=1025.655,-104.840,-87.950,166.583,45.947,158.380
C04440=1025.649,-105.090,-87.941,166.581,45.950,158.380
C04441=1025.643,-105.339,-87.932,166.577,45.952,158.380
C04442=1025.637,-105.589,-87.923,166.574,45.955,158.380
C04443=1025.632,-105.838,-87.913,166.572,45.958,158.381
C04444=1025.626,-106.088,-87.904,166.568,45.961,158.381
C04445=1025.620,-106.338,-87.895,166.566,45.963,158.381
C04446=1025.614,-106.587,-87.886,166.562,45.966,158.381
C04447=1025.609,-106.838,-87.876,166.559,45.969,158.381
C04448=1025.603,-107.087,-87.867,166.557,45.971,158.381
C04449=1025.598,-107.338,-87.858,166.553,45.974,158.381
C04450=1025.592,-107.587,-87.849,166.550,45.977,158.381
C04451=1025.586,-107.837,-87.840,166.547,45.979,158.382
C04452=1025.581,-108.086,-87.831,166.544,45.982,158.382
C04453=1025.574,-108.336,-87.822,166.542,45.985,158.382
C04454=1025.569,-108.586,-87.813,166.538,45.988,158.382
C04455=1025.563,-108.836,-87.803,166.535,45.991,158.382
C04456=1025.558,-109.085,-87.795,166.533,45.993,158.382
C04457=1025.552,-109.336,-87.786,166.529,45.996,158.382
C04458=1025.546,-109.585,-87.777,166.526,45.999,158.383
C04459=1025.540,-109.835,-87.768,166.524,46.002,158.383
C04460=1025.534,-110.084,-87.759,166.520,46.005,158.383
C04461=1025.528,-110.334,-87.751,166.517,46.008,158.383
C04462=1025.523,-110.584,-87.741,166.515,46.011,158.383
C04463=1025.517,-110.834,-87.733,166.511,46.013,158.383
C04464=1025.511,-111.084,-87.724,166.508,46.016,158.383
C04465=1025.505,-111.334,-87.715,166.505,46.019,158.384
C04466=1025.500,-111.583,-87.706,166.502,46.022,158.384
C04467=1025.494,-111.832,-87.697,166.499,46.025,158.384
C04468=1025.489,-112.083,-87.688,166.497,46.028,158.384
C04469=1025.483,-112.332,-87.680,166.493,46.030,158.384
C04470=1025.477,-112.582,-87.670,166.490,46.033,158.384
C04471=1025.472,-112.832,-87.661,166.487,46.036,158.385
C04472=1025.467,-113.082,-87.653,166.484,46.039,158.385
C04473=1025.460,-113.331,-87.643,166.481,46.042,158.385
C04474=1025.455,-113.581,-87.635,166.478,46.045,158.385
C04475=1025.449,-113.832,-87.626,166.475,46.047,158.385
C04476=1025.444,-114.081,-87.617,166.472,46.050,158.385
C04477=1025.438,-114.330,-87.608,166.469,46.053,158.385
C04478=1025.432,-114.581,-87.600,166.466,46.056,158.385
C04479=1025.427,-114.830,-87.592,166.464,46.059,158.386
C04480=1025.420,-115.080,-87.582,166.460,46.062,158.386
C04481=1025.415,-115.330,-87.574,166.457,46.065,158.386
C04482=1025.410,-115.579,-87.565,166.455,46.067,158.386
C04483=1025.404,-115.830,-87.556,166.451,46.070,158.386
C04484=1025.398,-116.079,-87.548,166.448,46.073,158.386
///RCONF 1,0,0,0,0,0,0,0,0,0,0,0,0,0,0,0,0,0,0,0,0,0,0,0
C04485=1025.392,-116.328,-87.539,166.445,46.075,158.387
C04486=1025.387,-116.579,-87.530,166.442,46.078,158.387
C04487=1025.380,-116.864,-87.520,166.439,46.082,158.387
C04488=1025.375,-117.150,-87.511,166.435,46.085,158.387
C04489=1025.368,-117.436,-87.501,166.431,46.088,158.387
C04490=1025.361,-117.721,-87.491,166.428,46.092,158.387
C04491=1025.356,-117.971,-87.483,166.425,46.095,158.388
C04492=1025.350,-118.222,-87.474,166.422,46.097,158.388
C04493=1025.344,-118.471,-87.466,166.419,46.100,158.388
C04494=1025.338,-118.721,-87.457,166.416,46.103,158.388
C04495=1025.333,-118.970,-87.449,166.413,46.106,158.388
C04496=1025.327,-119.221,-87.440,166.410,46.109,158.388
C04497=1025.321,-119.470,-87.432,166.407,46.112,158.388
C04498=1025.316,-119.720,-87.424,166.404,46.115,158.389
C04499=1025.310,-119.970,-87.414,166.401,46.118,158.389
C04500=1025.305,-120.219,-87.406,166.398,46.121,158.389
C04501=1025.299,-120.469,-87.398,166.396,46.124,158.389
C04502=1025.293,-120.719,-87.389,166.392,46.127,158.389
C04503=1025.287,-120.969,-87.380,166.389,46.130,158.389
C04504=1025.282,-121.219,-87.372,166.387,46.132,158.390
C04505=1025.276,-121.468,-87.364,166.383,46.135,158.390
C04506=1025.271,-121.718,-87.356,166.380,46.138,158.390
C04507=1025.266,-121.967,-87.347,166.378,46.141,158.390
C04508=1025.259,-122.218,-87.339,166.374,46.144,158.390
C04509=1025.254,-122.467,-87.330,166.371,46.147,158.390
C04510=1025.249,-122.718,-87.323,166.368,46.149,158.390
C04511=1025.243,-122.967,-87.315,166.365,46.152,158.390
C04512=1025.238,-123.217,-87.306,166.362,46.155,158.391
C04513=1025.232,-123.467,-87.297,166.360,46.158,158.391
C04514=1025.226,-123.717,-87.289,166.356,46.161,158.391
C04515=1025.220,-123.966,-87.281,166.353,46.164,158.391
C04516=1025.215,-124.216,-87.273,166.351,46.167,158.391
C04517=1025.210,-124.466,-87.264,166.347,46.170,158.391
C04518=1025.203,-124.716,-87.256,166.344,46.173,158.392
C04519=1025.198,-124.966,-87.248,166.341,46.176,158.392
C04520=1025.192,-125.216,-87.240,166.338,46.179,158.392
C04521=1025.187,-125.465,-87.232,166.335,46.182,158.392
C04522=1025.181,-125.715,-87.224,166.332,46.185,158.392
C04523=1025.176,-125.964,-87.215,166.329,46.188,158.392
C04524=1025.171,-126.215,-87.207,166.326,46.191,158.393
C04525=1025.164,-126.465,-87.199,166.323,46.194,158.393
C04526=1025.159,-126.715,-87.191,166.320,46.197,158.393
C04527=1025.153,-126.964,-87.183,166.317,46.200,158.393
C04528=1025.148,-127.214,-87.174,166.314,46.203,158.393
C04529=1025.142,-127.464,-87.167,166.310,46.206,158.393
C04530=1025.137,-127.713,-87.159,166.308,46.208,158.393
C04531=1025.131,-127.963,-87.151,166.305,46.212,158.394
C04532=1025.126,-128.213,-87.142,166.303,46.214,158.394
C04533=1025.122,-128.462,-87.134,166.299,46.217,158.394
C04534=1025.117,-128.712,-87.123,166.296,46.218,158.394
C04535=1025.114,-128.962,-87.112,166.294,46.218,158.394
C04536=1025.111,-129.211,-87.102,166.291,46.219,158.393
C04537=1025.109,-129.461,-87.090,166.289,46.220,158.393
C04538=1025.106,-129.710,-87.078,166.287,46.219,158.393
C04539=1025.106,-129.961,-87.066,166.284,46.218,158.392
C04540=1025.105,-130.210,-87.053,166.281,46.217,158.392
C04541=1025.105,-130.460,-87.039,166.279,46.215,158.391
C04542=1025.105,-130.709,-87.024,166.278,46.213,158.391
C04543=1025.106,-130.960,-87.010,166.275,46.210,158.390
C04544=1025.108,-131.209,-86.994,166.274,46.207,158.389
C04545=1025.109,-131.459,-86.977,166.271,46.203,158.388
C04546=1025.112,-131.709,-86.961,166.270,46.199,158.387
C04547=1025.114,-131.959,-86.943,166.268,46.194,158.387
C04548=1025.118,-132.209,-86.926,166.267,46.188,158.385
C04549=1025.122,-132.458,-86.907,166.265,46.183,158.384
C04550=1025.127,-132.708,-86.888,166.264,46.177,158.383
C04551=1024.827,-132.734,-87.219,166.216,46.449,158.423
C04552=1024.822,-132.484,-87.237,166.218,46.456,158.425
C04553=1024.818,-132.235,-87.256,166.219,46.462,158.426
C04554=1024.814,-131.985,-87.274,166.221,46.467,158.427
C04555=1024.811,-131.734,-87.292,166.221,46.471,158.428
C04556=1024.809,-131.485,-87.308,166.224,46.476,158.429
C04557=1024.807,-131.236,-87.324,166.226,46.479,158.429
C04558=1024.805,-130.986,-87.340,166.227,46.483,158.430
C04559=1024.805,-130.735,-87.355,166.229,46.485,158.431
C04560=1024.804,-130.486,-87.370,166.231,46.488,158.432
C04561=1024.804,-130.236,-87.383,166.234,46.490,158.432
C04562=1024.805,-129.986,-87.396,166.236,46.491,158.433
C04563=1024.807,-129.737,-87.409,166.238,46.492,158.433
C04564=1024.808,-129.487,-87.421,166.241,46.492,158.433
C04565=1024.811,-129.236,-87.432,166.243,46.492,158.433
C04566=1024.813,-128.987,-87.443,166.246,46.491,158.434
C04567=1024.817,-128.737,-87.454,166.249,46.490,158.434
C04568=1024.821,-128.488,-87.463,166.252,46.489,158.434
C04569=1024.826,-128.238,-87.472,166.254,46.487,158.434
C04570=1024.830,-127.988,-87.482,166.257,46.484,158.434
C04571=1024.836,-127.739,-87.489,166.260,46.481,158.434
C04572=1024.841,-127.489,-87.498,166.263,46.478,158.434
C04573=1024.847,-127.240,-87.506,166.266,46.475,158.433
C04574=1024.852,-126.989,-87.514,166.269,46.472,158.433
C04575=1024.858,-126.740,-87.521,166.272,46.469,158.433
C04576=1024.864,-126.490,-87.530,166.275,46.466,158.433
C04577=1024.870,-126.241,-87.538,166.278,46.463,158.433
C04578=1024.875,-125.991,-87.546,166.281,46.460,158.433
C04579=1024.881,-125.741,-87.553,166.284,46.457,158.433
C04580=1024.886,-125.491,-87.562,166.287,46.453,158.432
C04581=1024.892,-125.241,-87.571,166.290,46.450,158.432
C04582=1024.898,-124.992,-87.579,166.293,46.447,158.432
C04583=1024.903,-124.741,-87.586,166.296,46.444,158.432
C04584=1024.909,-124.492,-87.594,166.300,46.441,158.432
C04585=1024.914,-124.242,-87.603,166.302,46.438,158.431
C04586=1024.920,-123.992,-87.612,166.305,46.435,158.431
C04587=1024.926,-123.742,-87.620,166.308,46.432,158.431
C04588=1024.931,-123.493,-87.628,166.311,46.429,158.431
C04589=1024.936,-123.242,-87.636,166.314,46.426,158.431
C04590=1024.942,-122.993,-87.644,166.317,46.423,158.431
C04591=1024.947,-122.743,-87.652,166.321,46.420,158.431
C04592=1024.953,-122.493,-87.661,166.323,46.418,158.430
C04593=1024.958,-122.243,-87.670,166.326,46.414,158.430
C04594=1024.964,-121.994,-87.677,166.330,46.411,158.430
C04595=1024.970,-121.744,-87.686,166.332,46.409,158.430
C04596=1024.975,-121.494,-87.694,166.335,46.406,158.430
C04597=1024.982,-121.244,-87.703,166.338,46.403,158.430
C04598=1024.987,-120.994,-87.711,166.342,46.399,158.430
C04599=1024.992,-120.745,-87.720,166.344,46.397,158.429
C04600=1024.997,-120.495,-87.728,166.347,46.394,158.429
C04601=1025.003,-120.246,-87.736,166.351,46.391,158.429
C04602=1025.009,-119.995,-87.745,166.353,46.388,158.429
C04603=1025.014,-119.745,-87.753,166.356,46.385,158.429
C04604=1025.020,-119.496,-87.762,166.360,46.382,158.429
C04605=1025.026,-119.246,-87.770,166.363,46.379,158.428
C04606=1025.032,-118.996,-87.779,166.365,46.376,158.428
C04607=1025.037,-118.746,-87.787,166.368,46.373,158.428
C04608=1025.042,-118.496,-87.796,166.372,46.370,158.428
C04609=1025.048,-118.247,-87.803,166.374,46.367,158.428
C04610=1025.054,-117.997,-87.812,166.377,46.364,158.428
C04611=1025.060,-117.748,-87.822,166.381,46.361,158.428
C04612=1025.066,-117.461,-87.831,166.384,46.358,158.427
C04613=1025.073,-117.176,-87.841,166.387,46.354,158.427
C04614=1025.078,-116.891,-87.851,166.391,46.351,158.427
C04615=1025.085,-116.605,-87.861,166.395,46.348,158.427
C04616=1025.091,-116.355,-87.869,166.397,46.345,158.427
C04617=1025.097,-116.105,-87.877,166.400,46.342,158.427
C04618=1025.102,-115.855,-87.886,166.404,46.339,158.426
C04619=1025.108,-115.606,-87.894,166.407,46.336,158.426
C04620=1025.114,-115.355,-87.903,166.409,46.333,158.426
C04621=1025.119,-115.106,-87.912,166.412,46.330,158.426
C04622=1025.124,-114.856,-87.921,166.416,46.327,158.426
C04623=1025.131,-114.606,-87.929,166.418,46.324,158.426
C04624=1025.136,-114.357,-87.938,166.421,46.321,158.426
C04625=1025.142,-114.107,-87.947,166.425,46.318,158.425
C04626=1025.148,-113.857,-87.956,166.428,46.315,158.425
C04627=1025.153,-113.607,-87.964,166.430,46.312,158.425
C04628=1025.159,-113.357,-87.973,166.434,46.309,158.425
C04629=1025.164,-113.108,-87.982,166.437,46.306,158.425
C04630=1025.170,-112.858,-87.991,166.439,46.304,158.425
C04631=1025.176,-112.608,-88.000,166.443,46.301,158.425
C04632=1025.181,-112.359,-88.009,166.446,46.298,158.424
C04633=1025.187,-112.108,-88.018,166.448,46.295,158.424
C04634=1025.192,-111.859,-88.026,166.452,46.292,158.424
C04635=1025.198,-111.609,-88.035,166.455,46.289,158.424
C04636=1025.204,-111.359,-88.044,166.457,46.286,158.424
C04637=1025.210,-111.110,-88.052,166.461,46.283,158.424
C04638=1025.216,-110.860,-88.062,166.464,46.280,158.423
C04639=1025.221,-110.610,-88.070,166.466,46.278,158.423
C04640=1025.227,-110.360,-88.080,166.469,46.275,158.423
C04641=1025.233,-110.111,-88.088,166.473,46.272,158.423
C04642=1025.238,-109.860,-88.097,166.475,46.269,158.423
C04643=1025.244,-109.611,-88.106,166.479,46.266,158.423
C04644=1025.249,-109.361,-88.115,166.482,46.263,158.423
C04645=1025.255,-109.112,-88.124,166.485,46.260,158.423
C04646=1025.261,-108.862,-88.133,166.487,46.258,158.422
C04647=1025.267,-108.612,-88.142,166.491,46.255,158.422
C04648=1025.272,-108.362,-88.151,166.494,46.252,158.422
C04649=1025.278,-108.112,-88.160,166.496,46.249,158.422
C04650=1025.284,-107.863,-88.169,166.500,46.246,158.422
C04651=1025.289,-107.612,-88.178,166.503,46.243,158.422
C04652=1025.295,-107.363,-88.187,166.505,46.240,158.421
C04653=1025.301,-107.114,-88.196,166.509,46.238,158.421
C04654=1025.306,-106.864,-88.205,166.512,46.235,158.421
C04655=1025.313,-106.614,-88.215,166.514,46.232,158.421
C04656=1025.318,-106.364,-88.223,166.518,46.229,158.421
C04657=1025.324,-106.115,-88.233,166.521,46.226,158.421
C04658=1025.329,-105.864,-88.242,166.523,46.223,158.421
C04659=1025.335,-105.615,-88.251,166.527,46.221,158.421
C04660=1025.341,-105.365,-88.261,166.530,46.218,158.420
C04661=1025.346,-105.115,-88.269,166.533,46.215,158.420
C04662=1025.352,-104.865,-88.279,166.536,46.212,158.420
C04663=1025.358,-104.616,-88.288,166.539,46.209,158.420
C04664=1025.364,-104.366,-88.297,166.541,46.206,158.420
C04665=1025.369,-104.116,-88.307,166.545,46.204,158.420
C04666=1025.374,-103.866,-88.316,166.548,46.201,158.420
C04667=1025.381,-103.616,-88.325,166.551,46.198,158.419
C04668=1025.386,-103.367,-88.334,166.554,46.195,158.419
C04669=1025.392,-103.117,-88.344,166.557,46.192,158.419
C04670=1025.398,-102.867,-88.353,166.560,46.190,158.419
C04671=1025.404,-102.618,-88.362,166.563,46.187,158.419
C04672=1025.409,-102.368,-88.372,166.566,46.184,158.419
C04673=1025.415,-102.118,-88.381,166.569,46.181,158.418
C04674=1025.421,-101.868,-88.390,166.572,46.178,158.418
C04675=1025.427,-101.618,-88.400,166.574,46.175,158.418
C04676=1025.433,-101.333,-88.410,166.579,46.172,158.418
C04677=1025.440,-101.046,-88.421,166.582,46.169,158.418
C04678=1025.446,-100.761,-88.432,166.585,46.166,158.418
C04679=1025.452,-100.475,-88.443,166.589,46.163,158.418
C04680=1025.458,-100.225,-88.452,166.592,46.160,158.418
C04681=1025.464,-99.975,-88.461,166.595,46.157,158.417
C04682=1025.470,-99.725,-88.470,166.598,46.154,158.417
C04683=1025.476,-99.476,-88.480,166.601,46.151,158.417
C04684=1025.482,-99.226,-88.490,166.604,46.148,158.417
C04685=1025.488,-98.976,-88.500,166.607,46.146,158.417
C04686=1025.493,-98.727,-88.509,166.610,46.143,158.417
C04687=1025.499,-98.477,-88.518,166.612,46.140,158.416
C04688=1025.505,-98.226,-88.527,166.616,46.137,158.416
C04689=1025.511,-97.977,-88.537,166.619,46.134,158.416
C04690=1025.516,-97.727,-88.547,166.621,46.131,158.416
C04691=1025.522,-97.477,-88.556,166.625,46.129,158.416
C04692=1025.528,-97.227,-88.566,166.628,46.126,158.416
C04693=1025.533,-96.978,-88.576,166.630,46.123,158.416
C04694=1025.540,-96.728,-88.585,166.634,46.121,158.416
C04695=1025.545,-96.478,-88.595,166.636,46.118,158.415
C04696=1025.551,-96.229,-88.605,166.640,46.115,158.415
C04697=1025.556,-95.979,-88.615,166.643,46.113,158.415
C04698=1025.562,-95.729,-88.624,166.646,46.110,158.415
C04699=1025.568,-95.479,-88.634,166.649,46.107,158.415
C04700=1025.573,-95.230,-88.644,166.651,46.105,158.415
C04701=1025.579,-94.980,-88.654,166.655,46.102,158.415
C04702=1025.585,-94.730,-88.663,166.658,46.099,158.415
C04703=1025.590,-94.480,-88.674,166.661,46.097,158.414
C04704=1025.596,-94.231,-88.683,166.664,46.094,158.414
C04705=1025.602,-93.981,-88.694,166.666,46.091,158.414
C04706=1025.608,-93.732,-88.703,166.670,46.089,158.414
C04707=1025.613,-93.482,-88.713,166.672,46.086,158.414
C04708=1025.619,-93.232,-88.723,166.675,46.083,158.414
C04709=1025.624,-92.982,-88.733,166.679,46.081,158.414
C04710=1025.630,-92.733,-88.742,166.681,46.078,158.414
C04711=1025.636,-92.483,-88.752,166.685,46.075,158.413
C04712=1025.642,-92.233,-88.762,166.687,46.073,158.413
C04713=1025.648,-91.983,-88.772,166.690,46.070,158.413
C04714=1025.654,-91.733,-88.782,166.694,46.067,158.413
C04715=1025.659,-91.484,-88.792,166.696,46.065,158.413
C04716=1025.665,-91.234,-88.802,166.700,46.062,158.413
C04717=1025.671,-90.984,-88.811,166.702,46.059,158.413
C04718=1025.677,-90.735,-88.822,166.705,46.057,158.413
C04719=1025.683,-90.485,-88.832,166.709,46.054,158.412
C04720=1025.688,-90.235,-88.842,166.711,46.051,158.412
C04721=1025.694,-89.985,-88.852,166.714,46.048,158.412
C04722=1025.699,-89.736,-88.861,166.717,46.046,158.412
C04723=1025.706,-89.487,-88.872,166.720,46.043,158.412
C04724=1025.711,-89.236,-88.882,166.724,46.040,158.412
C04725=1025.717,-88.987,-88.891,166.726,46.038,158.412
C04726=1025.723,-88.737,-88.902,166.729,46.035,158.411
C04727=1025.729,-88.487,-88.912,166.732,46.032,158.411
C04728=1025.735,-88.237,-88.922,166.735,46.030,158.411
C04729=1025.741,-87.987,-88.932,166.739,46.027,158.411
C04730=1025.747,-87.738,-88.942,166.741,46.024,158.411
C04731=1025.753,-87.488,-88.952,166.744,46.021,158.411
C04732=1025.758,-87.238,-88.962,166.747,46.019,158.411
C04733=1025.764,-86.989,-88.973,166.750,46.016,158.411
C04734=1025.770,-86.740,-88.982,166.753,46.013,158.410
C04735=1025.775,-86.489,-88.992,166.756,46.011,158.410
C04736=1025.781,-86.240,-89.003,166.759,46.008,158.410
C04737=1025.787,-85.990,-89.013,166.762,46.005,158.410
C04738=1025.793,-85.740,-89.022,166.765,46.002,158.410
C04739=1025.799,-85.491,-89.033,166.769,46.000,158.410
C04740=1025.806,-85.206,-89.045,166.772,45.997,158.410
C04741=1025.812,-84.923,-89.056,166.775,45.993,158.409
C04742=1025.819,-84.639,-89.067,166.778,45.990,158.409
C04743=1025.826,-84.355,-89.080,166.782,45.987,158.409
C04744=1025.832,-84.105,-89.089,166.784,45.984,158.409
C04745=1025.838,-83.855,-89.100,166.787,45.982,158.409
C04746=1025.844,-83.606,-89.110,166.791,45.979,158.409
C04747=1025.850,-83.356,-89.120,166.793,45.976,158.408
C04748=1025.856,-83.106,-89.131,166.797,45.974,158.408
C04749=1025.862,-82.856,-89.140,166.800,45.971,158.408
C04750=1025.867,-82.607,-89.151,166.802,45.968,158.408
C04751=1025.874,-82.357,-89.161,166.806,45.965,158.408
C04752=1025.879,-82.108,-89.172,166.808,45.963,158.408
C04753=1025.886,-81.858,-89.181,166.811,45.960,158.408
C04754=1025.891,-81.608,-89.192,166.815,45.957,158.408
C04755=1025.897,-81.359,-89.202,166.817,45.954,158.407
C04756=1025.903,-81.109,-89.213,166.821,45.952,158.407
C04757=1025.909,-80.859,-89.222,166.823,45.949,158.407
C04758=1025.915,-80.610,-89.233,166.826,45.946,158.407
C04759=1025.921,-80.359,-89.244,166.830,45.943,158.407
C04760=1025.928,-80.110,-89.254,166.832,45.941,158.407
C04761=1025.933,-79.860,-89.264,166.835,45.938,158.407
C04762=1025.939,-79.610,-89.275,166.838,45.935,158.406
C04763=1025.945,-79.361,-89.286,166.841,45.933,158.406
C04764=1025.951,-79.111,-89.295,166.844,45.930,158.406
C04765=1025.956,-78.861,-89.306,166.847,45.928,158.406
C04766=1025.962,-78.612,-89.317,166.849,45.925,158.406
C04767=1025.968,-78.362,-89.327,166.853,45.922,158.406
C04768=1025.974,-78.112,-89.339,166.855,45.920,158.406
C04769=1025.980,-77.862,-89.349,166.859,45.917,158.405
C04770=1025.986,-77.613,-89.360,166.861,45.915,158.405
C04771=1025.992,-77.363,-89.370,166.865,45.912,158.405
C04772=1025.997,-77.113,-89.381,166.868,45.909,158.405
C04773=1026.003,-76.864,-89.392,166.870,45.907,158.405
C04774=1026.009,-76.614,-89.402,166.874,45.904,158.405
C04775=1026.016,-76.364,-89.412,166.876,45.902,158.405
C04776=1026.021,-76.114,-89.423,166.880,45.899,158.405
C04777=1026.027,-75.865,-89.434,166.882,45.896,158.404
C04778=1026.033,-75.615,-89.445,166.886,45.894,158.404
C04779=1026.038,-75.365,-89.455,166.888,45.891,158.404
C04780=1026.045,-75.115,-89.466,166.891,45.889,158.404
C04781=1026.051,-74.866,-89.477,166.894,45.886,158.404
C04782=1026.057,-74.616,-89.488,166.897,45.883,158.404
C04783=1026.063,-74.367,-89.498,166.900,45.881,158.404
C04784=1026.068,-74.117,-89.509,166.903,45.878,158.404
C04785=1026.074,-73.867,-89.520,166.905,45.876,158.403
C04786=1026.080,-73.617,-89.531,166.909,45.873,158.403
C04787=1026.086,-73.368,-89.542,166.911,45.871,158.403
C04788=1026.092,-73.118,-89.553,166.915,45.869,158.403
C04789=1026.097,-72.868,-89.564,166.917,45.866,158.403
C04790=1026.103,-72.618,-89.575,166.921,45.864,158.403
C04791=1026.109,-72.369,-89.586,166.923,45.861,158.403
C04792=1026.114,-72.119,-89.597,166.926,45.859,158.403
C04793=1026.120,-71.870,-89.608,166.929,45.856,158.403
C04794=1026.126,-71.620,-89.619,166.932,45.854,158.402
C04795=1026.132,-71.370,-89.630,166.935,45.852,158.402
C04796=1026.138,-71.121,-89.641,166.937,45.849,158.402
C04797=1026.143,-70.871,-89.652,166.941,45.847,158.402
C04798=1026.149,-70.621,-89.664,166.943,45.844,158.402
C04799=1026.155,-70.371,-89.674,166.947,45.842,158.402
C04800=1026.161,-70.122,-89.686,166.949,45.839,158.402
C04801=1026.167,-69.873,-89.697,166.953,45.837,158.402
C04802=1026.173,-69.623,-89.708,166.955,45.834,158.402
C04803=1026.179,-69.373,-89.719,166.958,45.832,158.401
C04804=1026.185,-69.091,-89.732,166.961,45.829,158.401
C04805=1026.192,-68.809,-89.744,166.965,45.827,158.401
C04806=1026.198,-68.528,-89.757,166.968,45.824,158.401
C04807=1026.205,-68.246,-89.769,166.971,45.821,158.401
C04808=1026.211,-67.996,-89.781,166.975,45.818,158.401
C04809=1026.217,-67.746,-89.792,166.977,45.816,158.401
C04810=1026.222,-67.497,-89.803,166.980,45.814,158.401
C04811=1026.229,-67.247,-89.814,166.983,45.811,158.400
C04812=1026.235,-66.998,-89.826,166.985,45.809,158.400
///RCONF 1,0,0,1,0,0,0,0,0,0,0,0,0,0,0,0,0,0,0,0,0,0,0,0
C04813=1026.240,-66.748,-89.836,166.989,45.806,158.400
C04814=1026.246,-66.498,-89.848,166.991,45.804,158.400
C04815=1026.252,-66.248,-89.859,166.995,45.801,158.400
C04816=1026.258,-65.999,-89.870,166.997,45.799,158.400
C04817=1026.264,-65.749,-89.882,167.001,45.796,158.400
C04818=1026.270,-65.500,-89.893,167.003,45.793,158.400
C04819=1026.276,-65.250,-89.904,167.005,45.791,158.399
C04820=1026.282,-65.000,-89.915,167.009,45.788,158.399
C04821=1026.287,-64.750,-89.926,167.011,45.786,158.399
C04822=1026.294,-64.501,-89.938,167.015,45.783,158.399
C04823=1026.299,-64.251,-89.949,167.017,45.781,158.399
C04824=1026.306,-64.001,-89.961,167.021,45.778,158.399
C04825=1026.311,-63.752,-89.971,167.023,45.776,158.399
C04826=1026.318,-63.503,-89.983,167.027,45.773,158.399
C04827=1026.323,-63.252,-89.995,167.029,45.771,158.398
C04828=1026.329,-63.003,-90.006,167.033,45.768,158.398
C04829=1026.336,-62.753,-90.018,167.035,45.766,158.398
C04830=1026.341,-62.504,-90.029,167.037,45.764,158.398
C04831=1026.348,-62.254,-90.040,167.041,45.761,158.398
C04832=1026.354,-62.005,-90.051,167.043,45.759,158.398
C04833=1026.359,-61.754,-90.063,167.047,45.756,158.398
C04834=1026.365,-61.505,-90.074,167.049,45.754,158.398
C04835=1026.371,-61.256,-90.086,167.053,45.751,158.398
C04836=1026.377,-61.006,-90.097,167.055,45.749,158.397
C04837=1026.383,-60.756,-90.108,167.058,45.746,158.397
C04838=1026.389,-60.506,-90.120,167.061,45.744,158.397
C04839=1026.395,-60.257,-90.131,167.064,45.741,158.397
C04840=1026.401,-60.007,-90.143,167.067,45.739,158.397
C04841=1026.407,-59.758,-90.154,167.070,45.736,158.397
C04842=1026.413,-59.507,-90.165,167.073,45.734,158.397
C04843=1026.419,-59.258,-90.177,167.075,45.731,158.396
C04844=1026.425,-59.008,-90.189,167.078,45.728,158.396
C04845=1026.432,-58.759,-90.201,167.081,45.726,158.396
C04846=1026.438,-58.509,-90.212,167.084,45.723,158.396
C04847=1026.444,-58.259,-90.224,167.087,45.721,158.396
C04848=1026.449,-58.010,-90.235,167.090,45.718,158.396
C04849=1026.455,-57.759,-90.246,167.093,45.716,158.396
C04850=1026.462,-57.511,-90.258,167.096,45.713,158.396
C04851=1026.468,-57.260,-90.269,167.099,45.711,158.395
C04852=1026.474,-57.012,-90.281,167.102,45.708,158.395
C04853=1026.480,-56.761,-90.293,167.104,45.705,158.395
C04854=1026.486,-56.511,-90.304,167.107,45.703,158.395
C04855=1026.492,-56.262,-90.315,167.110,45.700,158.395
C04856=1026.499,-56.012,-90.327,167.113,45.698,158.395
C04857=1026.505,-55.764,-90.339,167.116,45.695,158.395
C04858=1026.510,-55.513,-90.351,167.119,45.693,158.394
C04859=1026.517,-55.263,-90.363,167.122,45.690,158.394
C04860=1026.523,-55.014,-90.374,167.124,45.687,158.394
C04861=1026.529,-54.764,-90.386,167.128,45.685,158.394
C04862=1026.535,-54.514,-90.397,167.130,45.682,158.394
C04863=1026.541,-54.265,-90.409,167.133,45.680,158.394
C04864=1026.547,-54.015,-90.420,167.136,45.677,158.394
C04865=1026.554,-53.765,-90.432,167.139,45.675,158.393
C04866=1026.560,-53.516,-90.444,167.142,45.672,158.393
C04867=1026.566,-53.266,-90.456,167.144,45.670,158.393
C04868=1026.572,-52.986,-90.469,167.147,45.667,158.393
C04869=1026.580,-52.705,-90.481,167.151,45.664,158.393
C04870=1026.587,-52.425,-90.495,167.154,45.661,158.393
C04871=1026.593,-52.144,-90.508,167.158,45.658,158.393
C04872=1026.600,-51.895,-90.520,167.160,45.656,158.392
C04873=1026.606,-51.645,-90.532,167.163,45.653,158.392
C04874=1026.613,-51.395,-90.543,167.166,45.651,158.392
C04875=1026.618,-51.146,-90.555,167.169,45.648,158.392
C04876=1026.625,-50.896,-90.567,167.172,45.646,158.392
C04877=1026.631,-50.647,-90.579,167.175,45.643,158.392
C04878=1026.636,-50.397,-90.591,167.178,45.641,158.392
C04879=1026.642,-50.147,-90.603,167.180,45.638,158.391
C04880=1026.649,-49.897,-90.615,167.184,45.636,158.391
C04881=1026.655,-49.647,-90.628,167.186,45.634,158.391
C04882=1026.661,-49.399,-90.639,167.188,45.631,158.391
C04883=1026.666,-49.148,-90.651,167.192,45.629,158.391
C04884=1026.672,-48.898,-90.664,167.195,45.627,158.391
C04885=1026.678,-48.649,-90.675,167.197,45.624,158.391
C04886=1026.684,-48.399,-90.688,167.200,45.622,158.391
C04887=1026.690,-48.149,-90.700,167.203,45.620,158.391
C04888=1026.697,-47.900,-90.712,167.205,45.617,158.390
C04889=1026.702,-47.651,-90.725,167.209,45.615,158.390
C04890=1026.709,-47.401,-90.736,167.211,45.612,158.390
C04891=1026.715,-47.151,-90.749,167.214,45.610,158.390
C04892=1026.720,-46.902,-90.761,167.217,45.608,158.390
C04893=1026.727,-46.653,-90.773,167.220,45.605,158.390
C04894=1026.732,-46.403,-90.786,167.222,45.603,158.390
C04895=1026.738,-46.153,-90.798,167.226,45.600,158.389
C04896=1026.745,-45.903,-90.810,167.228,45.598,158.389
C04897=1026.750,-45.654,-90.822,167.231,45.596,158.389
C04898=1026.757,-45.404,-90.834,167.234,45.593,158.389
C04899=1026.763,-45.154,-90.846,167.237,45.591,158.389
C04900=1026.768,-44.904,-90.859,167.239,45.589,158.389
C04901=1026.775,-44.656,-90.871,167.242,45.586,158.389
C04902=1026.781,-44.406,-90.884,167.245,45.584,158.389
C04903=1026.787,-44.156,-90.896,167.247,45.581,158.388
C04904=1026.793,-43.906,-90.908,167.251,45.579,158.388
C04905=1026.799,-43.657,-90.921,167.253,45.576,158.388
C04906=1026.805,-43.407,-90.933,167.257,45.574,158.388
C04907=1026.811,-43.158,-90.945,167.259,45.572,158.388
C04908=1026.817,-42.908,-90.957,167.262,45.569,158.388
C04909=1026.823,-42.658,-90.970,167.265,45.567,158.388
C04910=1026.830,-42.408,-90.982,167.268,45.564,158.388
C04911=1026.836,-42.159,-90.995,167.270,45.562,158.387
C04912=1026.842,-41.909,-91.006,167.274,45.559,158.387
C04913=1026.848,-41.659,-91.019,167.276,45.557,158.387
C04914=1026.853,-41.410,-91.031,167.279,45.555,158.387
C04915=1026.860,-41.161,-91.044,167.282,45.552,158.387
C04916=1026.866,-40.911,-91.056,167.285,45.550,158.387
C04917=1026.872,-40.661,-91.069,167.287,45.547,158.387
C04918=1026.879,-40.412,-91.081,167.290,45.545,158.387
C04919=1026.885,-40.162,-91.093,167.293,45.542,158.386
C04920=1026.891,-39.912,-91.106,167.295,45.540,158.386
C04921=1026.897,-39.662,-91.118,167.299,45.538,158.386
C04922=1026.903,-39.413,-91.131,167.301,45.535,158.386
C04923=1026.909,-39.163,-91.144,167.303,45.533,158.386
C04924=1026.915,-38.914,-91.156,167.307,45.531,158.386
C04925=1026.921,-38.664,-91.168,167.310,45.528,158.386
C04926=1026.928,-38.415,-91.181,167.312,45.526,158.386
C04927=1026.933,-38.165,-91.194,167.315,45.524,158.385
C04928=1026.939,-37.915,-91.206,167.318,45.521,158.385
C04929=1026.945,-37.666,-91.219,167.321,45.519,158.385
C04930=1026.951,-37.416,-91.232,167.323,45.517,158.385
C04931=1026.957,-37.166,-91.245,167.327,45.514,158.385
C04932=1026.964,-36.886,-91.260,167.329,45.512,158.385
C04933=1026.971,-36.606,-91.273,167.332,45.510,158.385
C04934=1026.978,-36.326,-91.288,167.336,45.507,158.384
C04935=1026.984,-36.045,-91.302,167.338,45.505,158.384
C04936=1026.991,-35.796,-91.315,167.342,45.502,158.384
C04937=1026.997,-35.546,-91.328,167.344,45.500,158.384
C04938=1027.003,-35.297,-91.339,167.347,45.498,158.384
C04939=1027.009,-35.048,-91.353,167.349,45.495,158.384
C04940=1027.015,-34.798,-91.365,167.353,45.493,158.384
C04941=1027.021,-34.549,-91.379,167.355,45.491,158.384
C04942=1027.027,-34.299,-91.391,167.358,45.488,158.383
C04943=1027.033,-34.050,-91.404,167.360,45.486,158.383
C04944=1027.039,-33.800,-91.417,167.364,45.484,158.383
C04945=1027.045,-33.550,-91.429,167.366,45.481,158.383
C04946=1027.051,-33.301,-91.443,167.369,45.479,158.383
C04947=1027.057,-33.051,-91.455,167.371,45.477,158.383
C04948=1027.064,-32.801,-91.469,167.374,45.474,158.383
C04949=1027.070,-32.551,-91.482,167.377,45.472,158.383
C04950=1027.076,-32.302,-91.495,167.379,45.469,158.382
C04951=1027.082,-32.052,-91.507,167.383,45.467,158.382
C04952=1027.088,-31.803,-91.521,167.386,45.465,158.382
C04953=1027.094,-31.553,-91.533,167.388,45.462,158.382
C04954=1027.100,-31.304,-91.546,167.390,45.460,158.382
C04955=1027.107,-31.054,-91.558,167.394,45.458,158.382
C04956=1027.113,-30.805,-91.572,167.396,45.455,158.382
C04957=1027.119,-30.555,-91.584,167.399,45.453,158.382
C04958=1027.125,-30.306,-91.597,167.401,45.450,158.381
C04959=1027.131,-30.056,-91.610,167.405,45.448,158.381
C04960=1027.137,-29.806,-91.623,167.407,45.446,158.381
C04961=1027.144,-29.557,-91.637,167.410,45.444,158.381
C04962=1027.149,-29.307,-91.649,167.413,45.441,158.381
C04963=1027.156,-29.057,-91.663,167.416,45.439,158.381
C04964=1027.162,-28.807,-91.675,167.418,45.437,158.381
C04965=1027.168,-28.558,-91.689,167.421,45.435,158.380
C04966=1027.175,-28.309,-91.702,167.424,45.432,158.380
C04967=1027.180,-28.059,-91.714,167.427,45.430,158.380
C04968=1027.187,-27.810,-91.728,167.429,45.427,158.380
C04969=1027.193,-27.560,-91.740,167.431,45.425,158.380
C04970=1027.199,-27.311,-91.753,167.435,45.423,158.380
C04971=1027.206,-27.061,-91.767,167.437,45.420,158.380
C04972=1027.212,-26.811,-91.780,167.440,45.418,158.379
C04973=1027.217,-26.561,-91.794,167.442,45.416,158.379
C04974=1027.223,-26.312,-91.807,167.445,45.414,158.379
C04975=1027.229,-26.063,-91.820,167.448,45.411,158.379
C04976=1027.236,-25.813,-91.833,167.451,45.409,158.379
C04977=1027.241,-25.563,-91.847,167.453,45.407,158.379
C04978=1027.248,-25.313,-91.860,167.456,45.405,158.379
C04979=1027.254,-25.064,-91.873,167.458,45.402,158.379
C04980=1027.260,-24.815,-91.887,167.462,45.400,158.379
C04981=1027.266,-24.566,-91.900,167.465,45.398,158.378
C04982=1027.271,-24.315,-91.913,167.467,45.395,158.378
C04983=1027.278,-24.066,-91.926,167.469,45.393,158.378
C04984=1027.284,-23.816,-91.940,167.472,45.391,158.378
C04985=1027.291,-23.567,-91.953,167.476,45.389,158.378
C04986=1027.296,-23.317,-91.967,167.478,45.386,158.378
C04987=1027.302,-23.068,-91.980,167.480,45.384,158.378
C04988=1027.308,-22.818,-91.993,167.483,45.382,158.378
C04989=1027.315,-22.568,-92.007,167.485,45.379,158.377
C04990=1027.321,-22.319,-92.020,167.489,45.377,158.377
C04991=1027.327,-22.069,-92.034,167.491,45.375,158.377
C04992=1027.333,-21.820,-92.047,167.494,45.373,158.377
C04993=1027.339,-21.571,-92.060,167.496,45.371,158.377
C04994=1027.345,-21.320,-92.074,167.499,45.369,158.377
C04995=1027.352,-21.071,-92.088,167.503,45.366,158.377
C04996=1027.359,-20.790,-92.102,167.505,45.364,158.376
///RCONF 1,0,0,0,0,0,0,0,0,0,0,0,0,0,0,0,0,0,0,0,0,0,0,0
C04997=1027.365,-20.509,-92.118,167.508,45.361,158.376
C04998=1027.372,-20.228,-92.133,167.511,45.359,158.376
C04999=1027.379,-19.947,-92.148,167.514,45.356,158.376
C05000=1027.385,-19.697,-92.162,167.517,45.354,158.376
C05001=1027.391,-19.448,-92.175,167.519,45.351,158.376
C05002=1027.397,-19.199,-92.188,167.523,45.349,158.376
C05003=1027.404,-18.949,-92.202,167.525,45.347,158.375
C05004=1027.410,-18.699,-92.216,167.527,45.344,158.375
C05005=1027.416,-18.450,-92.229,167.530,45.342,158.375
C05006=1027.423,-18.200,-92.243,167.533,45.340,158.375
C05007=1027.429,-17.951,-92.256,167.536,45.337,158.375
C05008=1027.434,-17.701,-92.270,167.538,45.335,158.375
C05009=1027.441,-17.451,-92.283,167.541,45.333,158.375
C05010=1027.447,-17.202,-92.297,167.543,45.330,158.374
C05011=1027.453,-16.952,-92.310,167.546,45.328,158.374
C05012=1027.460,-16.702,-92.324,167.549,45.326,158.374
C05013=1027.466,-16.453,-92.337,167.552,45.323,158.374
C05014=1027.472,-16.204,-92.351,167.554,45.321,158.374
C05015=1027.479,-15.954,-92.366,167.557,45.319,158.374
C05016=1027.485,-15.705,-92.379,167.559,45.317,158.374
C05017=1027.491,-15.456,-92.392,167.562,45.315,158.373
C05018=1027.497,-15.205,-92.406,167.565,45.313,158.373
C05019=1027.503,-14.956,-92.420,167.568,45.310,158.373
C05020=1027.509,-14.707,-92.433,167.570,45.308,158.373
C05021=1027.515,-14.456,-92.448,167.573,45.306,158.373
C05022=1027.521,-14.208,-92.462,167.575,45.304,158.373
C05023=1027.527,-13.958,-92.476,167.578,45.301,158.373
C05024=1027.534,-13.708,-92.489,167.580,45.299,158.373
C05025=1027.539,-13.459,-92.503,167.584,45.297,158.373
C05026=1027.546,-13.210,-92.517,167.586,45.295,158.372
C05027=1027.552,-12.960,-92.531,167.589,45.293,158.372
C05028=1027.558,-12.710,-92.545,167.591,45.290,158.372
C05029=1027.564,-12.460,-92.559,167.594,45.288,158.372
C05030=1027.571,-12.211,-92.573,167.596,45.286,158.372
C05031=1027.576,-11.962,-92.587,167.599,45.284,158.372
C05032=1027.583,-11.712,-92.600,167.601,45.281,158.371
C05033=1027.588,-11.462,-92.614,167.605,45.279,158.371
C05034=1027.595,-11.213,-92.629,167.608,45.277,158.371
C05035=1027.601,-10.963,-92.642,167.610,45.275,158.371
C05036=1027.606,-10.714,-92.656,167.612,45.272,158.371
C05037=1027.613,-10.464,-92.671,167.615,45.270,158.371
C05038=1027.619,-10.215,-92.684,167.618,45.268,158.371
C05039=1027.626,-9.965,-92.698,167.620,45.266,158.371
C05040=1027.632,-9.716,-92.713,167.622,45.264,158.370
C05041=1027.638,-9.466,-92.726,167.626,45.262,158.370
C05042=1027.644,-9.216,-92.740,167.629,45.260,158.370
C05043=1027.650,-8.968,-92.754,167.631,45.257,158.370
C05044=1027.656,-8.718,-92.768,167.633,45.255,158.370
C05045=1027.662,-8.468,-92.782,167.636,45.253,158.370
C05046=1027.669,-8.219,-92.797,167.638,45.250,158.370
C05047=1027.675,-7.969,-92.810,167.641,45.248,158.370
C05048=1027.682,-7.720,-92.825,167.643,45.246,158.369
C05049=1027.687,-7.470,-92.839,167.647,45.243,158.369
C05050=1027.694,-7.220,-92.852,167.649,45.241,158.369
C05051=1027.700,-6.971,-92.867,167.652,45.239,158.369
C05052=1027.706,-6.721,-92.881,167.654,45.237,158.369
C05053=1027.712,-6.472,-92.895,167.657,45.235,158.369
C05054=1027.718,-6.222,-92.909,167.659,45.233,158.369
C05055=1027.725,-5.973,-92.923,167.662,45.230,158.368
C05056=1027.731,-5.723,-92.938,167.664,45.228,158.368
C05057=1027.737,-5.474,-92.951,167.668,45.226,158.368
C05058=1027.744,-5.224,-92.966,167.670,45.223,158.368
C05059=1027.749,-4.975,-92.980,167.673,45.221,158.368
C05060=1027.757,-4.692,-92.996,167.675,45.218,158.368
C05061=1027.764,-4.409,-93.012,167.679,45.216,158.368
C05062=1027.771,-4.127,-93.027,167.681,45.213,158.367
C05063=1027.778,-3.845,-93.044,167.684,45.210,158.367
C05064=1027.784,-3.595,-93.059,167.687,45.208,158.367
C05065=1027.790,-3.345,-93.073,167.689,45.206,158.367
C05066=1027.796,-3.096,-93.088,167.692,45.204,158.367
C05067=1027.803,-2.846,-93.102,167.695,45.202,158.367
C05068=1027.808,-2.597,-93.116,167.697,45.200,158.367
C05069=1027.815,-2.347,-93.131,167.700,45.198,158.366
C05070=1027.820,-2.098,-93.145,167.702,45.196,158.366
C05071=1027.827,-1.848,-93.160,167.705,45.194,158.366
C05072=1027.833,-1.599,-93.174,167.707,45.192,158.366
C05073=1027.839,-1.349,-93.189,167.710,45.190,158.366
C05074=1027.844,-1.100,-93.203,167.712,45.188,158.366
C05075=1027.851,-0.850,-93.218,167.715,45.186,158.366
C05076=1027.857,-0.601,-93.233,167.717,45.183,158.365
C05077=1027.863,-0.351,-93.247,167.721,45.181,158.365
C05078=1027.869,-0.101,-93.262,167.723,45.179,158.365
C05079=1027.876,0.147,-93.276,167.726,45.177,158.365
C05080=1027.882,0.397,-93.291,167.729,45.175,158.365
C05081=1027.887,0.647,-93.305,167.731,45.173,158.365
C05082=1027.894,0.896,-93.320,167.733,45.170,158.365
C05083=1027.900,1.146,-93.335,167.736,45.168,158.365
C05084=1027.906,1.395,-93.349,167.739,45.166,158.364
C05085=1027.912,1.645,-93.363,167.741,45.164,158.364
C05086=1027.918,1.894,-93.378,167.744,45.162,158.364
C05087=1027.924,2.144,-93.393,167.746,45.160,158.364
C05088=1027.931,2.393,-93.408,167.749,45.158,158.364
C05089=1027.936,2.642,-93.423,167.751,45.156,158.364
C05090=1027.942,2.893,-93.437,167.754,45.154,158.364
C05091=1027.949,3.142,-93.452,167.756,45.151,158.363
C05092=1027.955,3.391,-93.466,167.759,45.149,158.363
C05093=1027.961,3.641,-93.481,167.761,45.147,158.363
C05094=1027.967,3.891,-93.496,167.764,45.145,158.363
C05095=1027.973,4.140,-93.511,167.766,45.143,158.363
C05096=1027.980,4.389,-93.525,167.769,45.140,158.363
C05097=1027.986,4.639,-93.539,167.771,45.138,158.363
C05098=1027.992,4.888,-93.554,167.774,45.136,158.363
C05099=1027.998,5.138,-93.569,167.776,45.134,158.362
C05100=1028.005,5.387,-93.584,167.779,45.132,158.362
C05101=1028.011,5.636,-93.598,167.781,45.130,158.362
C05102=1028.017,5.886,-93.613,167.785,45.127,158.362
C05103=1028.023,6.136,-93.628,167.787,45.125,158.362
C05104=1028.029,6.385,-93.643,167.790,45.123,158.362
C05105=1028.036,6.634,-93.658,167.792,45.121,158.362
C05106=1028.042,6.884,-93.673,167.795,45.119,158.361
C05107=1028.048,7.134,-93.688,167.797,45.116,158.361
C05108=1028.054,7.383,-93.702,167.800,45.114,158.361
C05109=1028.060,7.633,-93.717,167.802,45.112,158.361
C05110=1028.067,7.883,-93.731,167.805,45.110,158.361
C05111=1028.072,8.131,-93.746,167.807,45.107,158.361
C05112=1028.079,8.381,-93.761,167.810,45.105,158.361
C05113=1028.085,8.631,-93.776,167.812,45.103,158.360
C05114=1028.092,8.880,-93.791,167.815,45.101,158.360
C05115=1028.098,9.130,-93.806,167.817,45.099,158.360
C05116=1028.104,9.379,-93.820,167.820,45.097,158.360
C05117=1028.110,9.629,-93.835,167.822,45.094,158.360
C05118=1028.116,9.878,-93.850,167.825,45.092,158.360
C05119=1028.123,10.128,-93.865,167.827,45.090,158.359
C05120=1028.129,10.377,-93.880,167.830,45.087,158.359
C05121=1028.135,10.626,-93.895,167.832,45.085,158.359
C05122=1028.142,10.876,-93.910,167.835,45.083,158.359
C05123=1028.148,11.125,-93.925,167.837,45.081,158.359
C05124=1028.155,11.410,-93.941,167.841,45.079,158.359
C05125=1028.162,11.695,-93.959,167.843,45.076,158.358
C05126=1028.170,11.979,-93.975,167.846,45.073,158.358
C05127=1028.177,12.263,-93.993,167.849,45.071,158.358
C05128=1028.183,12.513,-94.008,167.851,45.068,158.358
C05129=1028.190,12.763,-94.023,167.854,45.066,158.358
C05130=1028.196,13.012,-94.038,167.857,45.064,158.358
C05131=1028.202,13.261,-94.053,167.860,45.061,158.357
C05132=1028.209,13.510,-94.068,167.862,45.060,158.357
C05133=1028.215,13.760,-94.083,167.865,45.058,158.357
C05134=1028.221,14.010,-94.098,167.867,45.055,158.357
C05135=1028.227,14.260,-94.113,167.870,45.053,158.357
C05136=1028.233,14.509,-94.128,167.872,45.051,158.357
C05137=1028.239,14.758,-94.143,167.875,45.049,158.357
C05138=1028.246,15.007,-94.158,167.877,45.047,158.357
C05139=1028.252,15.257,-94.174,167.880,45.044,158.356
C05140=1028.258,15.507,-94.189,167.882,45.042,158.356
C05141=1028.265,15.756,-94.205,167.885,45.040,158.356
C05142=1028.270,16.006,-94.220,167.888,45.038,158.356
C05143=1028.277,16.256,-94.235,167.890,45.036,158.356
C05144=1028.283,16.504,-94.250,167.891,45.034,158.355
C05145=1028.289,16.754,-94.265,167.894,45.032,158.355
C05146=1028.295,17.004,-94.281,167.897,45.030,158.355
C05147=1028.301,17.253,-94.296,167.899,45.028,158.355
C05148=1028.308,17.502,-94.311,167.901,45.025,158.355
C05149=1028.314,17.752,-94.326,167.904,45.023,158.355
C05150=1028.320,18.001,-94.343,167.907,45.021,158.355
C05151=1028.327,18.251,-94.358,167.909,45.019,158.354
C05152=1028.332,18.500,-94.372,167.911,45.017,158.354
C05153=1028.339,18.749,-94.388,167.914,45.015,158.354
C05154=1028.345,18.999,-94.403,167.917,45.013,158.354
C05155=1028.351,19.248,-94.418,167.919,45.010,158.354
C05156=1028.358,19.498,-94.434,167.922,45.008,158.354
C05157=1028.363,19.747,-94.450,167.924,45.006,158.354
C05158=1028.370,19.997,-94.465,167.927,45.004,158.353
C05159=1028.376,20.246,-94.480,167.929,45.002,158.353
C05160=1028.382,20.496,-94.496,167.932,44.999,158.353
C05161=1028.389,20.745,-94.511,167.934,44.997,158.353
C05162=1028.394,20.995,-94.527,167.937,44.995,158.353
C05163=1028.401,21.244,-94.543,167.939,44.993,158.353
C05164=1028.407,21.494,-94.558,167.942,44.991,158.353
C05165=1028.413,21.742,-94.573,167.944,44.989,158.352
C05166=1028.419,21.992,-94.588,167.947,44.987,158.352
C05167=1028.425,22.242,-94.605,167.949,44.985,158.352
C05168=1028.432,22.491,-94.620,167.952,44.983,158.352
C05169=1028.438,22.741,-94.636,167.954,44.980,158.352
C05170=1028.444,22.990,-94.651,167.957,44.978,158.352
C05171=1028.450,23.240,-94.667,167.959,44.976,158.352
C05172=1028.456,23.489,-94.682,167.962,44.974,158.351
C05173=1028.463,23.738,-94.698,167.964,44.972,158.351
C05174=1028.469,23.988,-94.714,167.967,44.970,158.351
C05175=1028.475,24.237,-94.729,167.969,44.968,158.351
C05176=1028.481,24.487,-94.745,167.972,44.966,158.351
C05177=1028.488,24.736,-94.760,167.973,44.963,158.351
C05178=1028.494,24.986,-94.776,167.976,44.961,158.350
C05179=1028.500,25.235,-94.791,167.978,44.959,158.350
C05180=1028.507,25.484,-94.807,167.981,44.957,158.350
C05181=1028.513,25.734,-94.823,167.983,44.955,158.350
C05182=1028.519,25.983,-94.838,167.986,44.953,158.350
C05183=1028.525,26.233,-94.854,167.988,44.951,158.350
C05184=1028.531,26.482,-94.869,167.991,44.949,158.350
C05185=1028.537,26.732,-94.886,167.993,44.946,158.349
C05186=1028.544,26.981,-94.901,167.996,44.944,158.349
C05187=1028.550,27.231,-94.917,167.999,44.942,158.349
C05188=1028.558,27.517,-94.935,168.001,44.939,158.349
C05189=1028.564,27.802,-94.953,168.004,44.937,158.349
C05190=1028.571,28.088,-94.971,168.007,44.935,158.349
C05191=1028.579,28.374,-94.990,168.010,44.932,158.348
C05192=1028.585,28.624,-95.005,168.012,44.930,158.348
C05193=1028.591,28.873,-95.021,168.014,44.928,158.348
C05194=1028.597,29.122,-95.037,168.017,44.926,158.348
C05195=1028.604,29.371,-95.053,168.019,44.924,158.348
C05196=1028.609,29.621,-95.069,168.022,44.922,158.348
C05197=1028.615,29.871,-95.085,168.025,44.920,158.348
C05198=1028.622,30.120,-95.101,168.027,44.917,158.347
C05199=1028.628,30.369,-95.117,168.029,44.915,158.347
C05200=1028.634,30.618,-95.133,168.032,44.913,158.347
C05201=1028.640,30.868,-95.148,168.035,44.911,158.347
C05202=1028.646,31.117,-95.164,168.037,44.909,158.347
C05203=1028.652,31.367,-95.181,168.040,44.907,158.347
C05204=1028.659,31.616,-95.196,168.041,44.905,158.346
C05205=1028.665,31.865,-95.212,168.044,44.903,158.346
C05206=1028.671,32.115,-95.229,168.046,44.901,158.346
C05207=1028.678,32.364,-95.245,168.049,44.898,158.346
C05208=1028.684,32.614,-95.260,168.051,44.896,158.346
C05209=1028.690,32.863,-95.277,168.054,44.895,158.346
C05210=1028.696,33.113,-95.293,168.056,44.893,158.346
C05211=1028.702,33.362,-95.308,168.059,44.891,158.345
C05212=1028.708,33.611,-95.325,168.061,44.888,158.345
C05213=1028.714,33.861,-95.341,168.064,44.886,158.345
C05214=1028.721,34.110,-95.357,168.066,44.884,158.345
C05215=1028.727,34.360,-95.373,168.069,44.882,158.345
C05216=1028.733,34.609,-95.389,168.071,44.879,158.345
C05217=1028.740,34.858,-95.405,168.073,44.878,158.344
C05218=1028.746,35.108,-95.421,168.075,44.876,158.344
C05219=1028.752,35.357,-95.437,168.078,44.874,158.344
C05220=1028.758,35.606,-95.453,168.080,44.871,158.344
C05221=1028.765,35.856,-95.469,168.083,44.869,158.344
C05222=1028.771,36.106,-95.485,168.085,44.867,158.344
C05223=1028.777,36.355,-95.502,168.088,44.864,158.343
C05224=1028.783,36.604,-95.517,168.090,44.862,158.343
C05225=1028.789,36.853,-95.534,168.093,44.860,158.343
C05226=1028.795,37.103,-95.550,168.095,44.859,158.343
C05227=1028.802,37.353,-95.567,168.098,44.856,158.343
C05228=1028.808,37.582,-95.582,168.099,44.854,158.343
C05229=1028.813,37.811,-95.596,168.102,44.853,158.343
C05230=1028.819,38.040,-95.611,168.105,44.851,158.343
C05231=1028.824,38.271,-95.627,168.106,44.849,158.342
C05232=1028.830,38.500,-95.642,168.109,44.847,158.342
C05233=1028.836,38.729,-95.656,168.111,44.845,158.342
C05234=1028.842,38.958,-95.672,168.113,44.843,158.342
C05235=1028.848,39.189,-95.686,168.116,44.841,158.342
C05236=1028.854,39.438,-95.703,168.118,44.839,158.342
C05237=1028.860,39.687,-95.720,168.121,44.837,158.341
C05238=1028.866,39.936,-95.736,168.123,44.835,158.341
C05239=1028.872,40.185,-95.752,168.126,44.833,158.341
C05240=1028.878,40.435,-95.769,168.127,44.831,158.341
C05241=1028.884,40.685,-95.785,168.130,44.828,158.341
C05242=1028.890,40.934,-95.801,168.132,44.826,158.341
C05243=1028.897,41.183,-95.818,168.135,44.825,158.341
C05244=1028.903,41.432,-95.835,168.137,44.823,158.340
C05245=1028.909,41.682,-95.851,168.140,44.821,158.340
C05246=1028.915,41.932,-95.867,168.142,44.818,158.340
C05247=1028.921,42.181,-95.884,168.145,44.816,158.340
C05248=1028.927,42.430,-95.900,168.147,44.814,158.340
C05249=1028.934,42.680,-95.917,168.149,44.812,158.340
C05250=1028.940,42.929,-95.933,168.151,44.810,158.339
C05251=1028.946,43.178,-95.950,168.154,44.808,158.339
C05252=1028.954,43.504,-95.972,168.157,44.805,158.339
C05253=1028.962,43.829,-95.994,168.161,44.803,158.339
C05254=1028.970,44.156,-96.015,168.163,44.800,158.339
C05255=1028.977,44.481,-96.037,168.167,44.798,158.339
C05256=1028.983,44.730,-96.053,168.169,44.796,158.339
C05257=1028.990,44.980,-96.071,168.172,44.794,158.338
C05258=1028.996,45.229,-96.087,168.173,44.791,158.338
C05259=1029.002,45.478,-96.104,168.176,44.789,158.338
C05260=1029.007,45.727,-96.121,168.178,44.788,158.338
C05261=1029.014,45.977,-96.138,168.181,44.786,158.338
C05262=1029.020,46.226,-96.155,168.183,44.784,158.338
C05263=1029.026,46.476,-96.171,168.186,44.782,158.337
C05264=1029.033,46.725,-96.188,168.189,44.780,158.337
C05265=1029.038,46.975,-96.205,168.190,44.778,158.337
C05266=1029.044,47.224,-96.221,168.193,44.776,158.337
C05267=1029.050,47.473,-96.238,168.195,44.774,158.337
C05268=1029.057,47.723,-96.255,168.198,44.771,158.337
C05269=1029.063,47.972,-96.272,168.200,44.769,158.337
C05270=1029.069,48.221,-96.289,168.203,44.767,158.336
C05271=1029.075,48.471,-96.306,168.204,44.766,158.336
C05272=1029.081,48.720,-96.322,168.207,44.764,158.336
C05273=1029.088,48.969,-96.339,168.210,44.762,158.336
C05274=1029.093,49.219,-96.356,168.212,44.760,158.336
C05275=1029.100,49.468,-96.373,168.214,44.757,158.336
C05276=1029.106,49.717,-96.390,168.217,44.755,158.335
C05277=1029.112,49.967,-96.407,168.220,44.753,158.335
C05278=1029.118,50.216,-96.424,168.221,44.751,158.335
C05279=1029.124,50.465,-96.441,168.224,44.750,158.335
C05280=1029.130,50.715,-96.457,168.226,44.748,158.335
C05281=1029.137,50.964,-96.474,168.229,44.745,158.335
C05282=1029.142,51.213,-96.491,168.231,44.743,158.335
C05283=1029.149,51.463,-96.509,168.234,44.741,158.334
C05284=1029.155,51.712,-96.525,168.236,44.739,158.334
C05285=1029.162,51.962,-96.542,168.239,44.737,158.334
C05286=1029.167,52.211,-96.559,168.240,44.735,158.334
C05287=1029.173,52.460,-96.576,168.243,44.733,158.334
C05288=1029.180,52.710,-96.593,168.245,44.731,158.334
C05289=1029.186,52.959,-96.610,168.248,44.729,158.334
C05290=1029.191,53.208,-96.627,168.251,44.727,158.333
C05291=1029.198,53.458,-96.644,168.253,44.725,158.333
C05292=1029.204,53.707,-96.661,168.255,44.722,158.333
C05293=1029.211,53.957,-96.677,168.257,44.720,158.333
C05294=1029.216,54.206,-96.695,168.260,44.719,158.333
C05295=1029.223,54.455,-96.712,168.262,44.717,158.333
C05296=1029.229,54.704,-96.729,168.265,44.714,158.332
C05297=1029.235,54.953,-96.746,168.267,44.712,158.332
C05298=1029.241,55.203,-96.763,168.270,44.710,158.332
C05299=1029.247,55.452,-96.780,168.272,44.708,158.332
C05300=1029.254,55.702,-96.797,168.275,44.706,158.332
C05301=1029.261,55.950,-96.814,168.276,44.704,158.331
C05302=1029.266,56.201,-96.831,168.279,44.702,158.331
C05303=1029.273,56.449,-96.848,168.281,44.700,158.331
C05304=1029.279,56.699,-96.866,168.284,44.698,158.331
C05305=1029.285,56.948,-96.882,168.286,44.695,158.331
C05306=1029.292,57.198,-96.900,168.289,44.693,158.331
C05307=1029.298,57.447,-96.917,168.291,44.691,158.331
C05308=1029.304,57.697,-96.933,168.294,44.689,158.330
C05309=1029.311,57.946,-96.950,168.296,44.687,158.330
C05310=1029.317,58.195,-96.968,168.298,44.685,158.330
C05311=1029.323,58.444,-96.985,168.300,44.683,158.330
C05312=1029.330,58.694,-97.002,168.303,44.680,158.330
C05313=1029.335,58.943,-97.019,168.305,44.678,158.329
C05314=1029.342,59.193,-97.037,168.308,44.676,158.329
C05315=1029.348,59.441,-97.054,168.311,44.675,158.329
C05316=1029.355,59.727,-97.074,168.313,44.672,158.329
C05317=1029.363,60.013,-97.093,168.316,44.669,158.329
C05318=1029.369,60.298,-97.113,168.319,44.667,158.329
C05319=1029.377,60.584,-97.132,168.321,44.664,158.328
C05320=1029.384,60.833,-97.149,168.324,44.663,158.328
C05321=1029.389,61.082,-97.167,168.326,44.660,158.328
C05322=1029.396,61.332,-97.184,168.329,44.658,158.328
C05323=1029.402,61.581,-97.200,168.331,44.656,158.328
C05324=1029.409,61.830,-97.218,168.334,44.653,158.327
C05325=1029.414,62.079,-97.235,168.336,44.651,158.327
C05326=1029.421,62.329,-97.253,168.339,44.649,158.327
C05327=1029.428,62.577,-97.270,168.340,44.647,158.327
C05328=1029.434,62.827,-97.288,168.343,44.645,158.327
C05329=1029.440,63.077,-97.304,168.345,44.643,158.327
C05330=1029.447,63.326,-97.321,168.348,44.641,158.326
C05331=1029.453,63.576,-97.339,168.350,44.639,158.326
C05332=1029.459,63.824,-97.356,168.353,44.637,158.326
C05333=1029.465,64.074,-97.374,168.355,44.635,158.326
C05334=1029.471,64.323,-97.391,168.358,44.633,158.326
C05335=1029.477,64.573,-97.409,168.359,44.630,158.326
C05336=1029.484,64.822,-97.427,168.362,44.628,158.325
C05337=1029.490,65.071,-97.444,168.364,44.626,158.325
C05338=1029.496,65.321,-97.462,168.367,44.624,158.325
C05339=1029.502,65.570,-97.479,168.369,44.623,158.325
C05340=1029.508,65.819,-97.497,168.372,44.620,158.325
C05341=1029.515,66.069,-97.514,168.374,44.618,158.325
C05342=1029.521,66.318,-97.532,168.376,44.616,158.324
C05343=1029.527,66.568,-97.550,168.379,44.614,158.324
C05344=1029.533,66.816,-97.566,168.381,44.612,158.324
C05345=1029.539,67.066,-97.584,168.383,44.610,158.324
C05346=1029.545,67.315,-97.602,168.386,44.608,158.324
C05347=1029.552,67.564,-97.620,168.389,44.606,158.324
C05348=1029.558,67.814,-97.638,168.391,44.604,158.324
C05349=1029.564,68.062,-97.655,168.393,44.602,158.323
C05350=1029.570,68.312,-97.673,168.395,44.600,158.323
C05351=1029.576,68.562,-97.691,168.398,44.598,158.323
C05352=1029.583,68.811,-97.708,168.400,44.596,158.323
C05353=1029.589,69.060,-97.726,168.403,44.594,158.323
C05354=1029.594,69.309,-97.743,168.405,44.592,158.323
C05355=1029.600,69.559,-97.761,168.408,44.590,158.322
C05356=1029.608,69.808,-97.779,168.410,44.588,158.322
C05357=1029.613,70.057,-97.797,168.412,44.585,158.322
C05358=1029.619,70.307,-97.815,168.414,44.583,158.322
C05359=1029.625,70.556,-97.833,168.417,44.582,158.322
C05360=1029.632,70.805,-97.850,168.420,44.580,158.322
C05361=1029.638,71.054,-97.868,168.422,44.578,158.321
C05362=1029.644,71.304,-97.886,168.424,44.576,158.321
C05363=1029.650,71.553,-97.904,168.426,44.573,158.321
C05364=1029.656,71.803,-97.922,168.429,44.571,158.321
C05365=1029.663,72.052,-97.940,168.431,44.569,158.321
C05366=1029.669,72.301,-97.957,168.434,44.567,158.321
C05367=1029.675,72.550,-97.975,168.436,44.566,158.321
C05368=1029.681,72.800,-97.993,168.438,44.564,158.320
C05369=1029.687,73.049,-98.012,168.441,44.562,158.320
C05370=1029.693,73.298,-98.029,168.443,44.559,158.320
C05371=1029.700,73.548,-98.047,168.446,44.557,158.320
C05372=1029.705,73.796,-98.065,168.448,44.555,158.320
C05373=1029.712,74.046,-98.083,168.451,44.553,158.320
C05374=1029.718,74.296,-98.101,168.453,44.551,158.319
C05375=1029.724,74.544,-98.119,168.455,44.549,158.319
C05376=1029.730,74.793,-98.137,168.457,44.547,158.319
C05377=1029.736,75.043,-98.155,168.460,44.545,158.319
C05378=1029.743,75.292,-98.173,168.462,44.543,158.319
C05379=1029.748,75.541,-98.191,168.465,44.541,158.319
C05380=1029.756,75.827,-98.211,168.467,44.539,158.318
C05381=1029.763,76.112,-98.232,168.470,44.537,158.318
C05382=1029.770,76.397,-98.253,168.473,44.534,158.318
C05383=1029.777,76.683,-98.273,168.476,44.532,158.318
C05384=1029.784,76.932,-98.291,168.478,44.530,158.318
C05385=1029.789,77.181,-98.309,168.481,44.527,158.317
C05386=1029.796,77.431,-98.328,168.482,44.526,158.317
C05387=1029.802,77.680,-98.345,168.485,44.524,158.317
C05388=1029.808,77.929,-98.364,168.487,44.522,158.317
C05389=1029.814,78.178,-98.382,168.490,44.520,158.317
C05390=1029.820,78.428,-98.400,168.493,44.518,158.317
C05391=1029.826,78.677,-98.418,168.495,44.516,158.317
C05392=1029.833,78.926,-98.437,168.497,44.514,158.316
C05393=1029.838,79.175,-98.454,168.499,44.512,158.316
C05394=1029.845,79.425,-98.473,168.502,44.510,158.316
C05395=1029.850,79.675,-98.492,168.504,44.508,158.316
C05396=1029.856,79.923,-98.510,168.507,44.506,158.316
C05397=1029.862,80.173,-98.528,168.509,44.504,158.316
C05398=1029.868,80.422,-98.547,168.511,44.502,158.315
C05399=1029.875,80.671,-98.565,168.514,44.500,158.315
C05400=1029.881,80.921,-98.583,168.516,44.498,158.315
C05401=1029.887,81.169,-98.601,168.519,44.496,158.315
C05402=1029.893,81.419,-98.619,168.521,44.494,158.315
C05403=1029.899,81.668,-98.638,168.524,44.492,158.315
C05404=1029.906,81.917,-98.657,168.525,44.490,158.314
C05405=1029.911,82.166,-98.674,168.528,44.488,158.314
C05406=1029.917,82.416,-98.693,168.530,44.486,158.314
C05407=1029.923,82.665,-98.711,168.533,44.484,158.314
